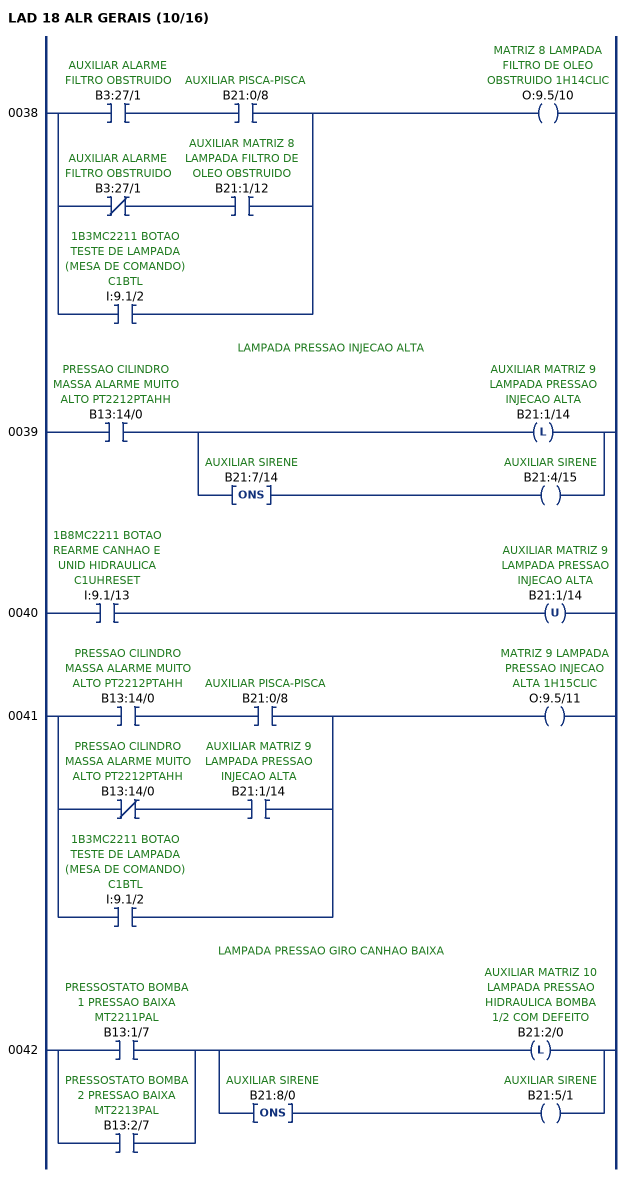
% Rung: 38 %
SOR BST XIC B3:27/1 XIC B21:0/8 NXB XIO B3:27/1 XIC B21:1/12 NXB XIC I:9.1/2 BND OTE O:9.5/10 EOR
%   B3:27/1  "AUXILIAR ALARME FILTRO OBSTRUIDO" %
%   B21:0/8  "AUXILIAR PISCA-PISCA" %
%   B21:1/12  "AUXILIAR MATRIZ 8 LAMPADA FILTRO DE OLEO OBSTRUIDO" %
%   I:9.1/2  C1BTL  "1B3MC2211 BOTAO TESTE DE LAMPADA (MESA DE COMANDO)" %
%   O:9.5/10  1H14CLIC  "MATRIZ 8 LAMPADA FILTRO DE OLEO OBSTRUIDO" %
% Rung: 39 %
% LAMPADA PRESSAO INJECAO ALTA %
SOR XIC B13:14/0 BST OTL B21:1/14 NXB OSR B21:7/14 OTE B21:4/15 BND EOR
%   B13:14/0  PT2212PTAHH  "PRESSAO CILINDRO MASSA ALARME MUITO ALTO" %
%   B21:1/14  "AUXILIAR MATRIZ 9 LAMPADA PRESSAO INJECAO ALTA" %
%   B21:7/14  "AUXILIAR SIRENE" %
%   B21:4/15  "AUXILIAR SIRENE" %
% Rung: 40 %
SOR XIC I:9.1/13 OTU B21:1/14 EOR
%   I:9.1/13  C1UHRESET  "1B8MC2211 BOTAO REARME CANHAO E UNID HIDRAULICA" %
%   B21:1/14  "AUXILIAR MATRIZ 9 LAMPADA PRESSAO INJECAO ALTA" %
% Rung: 41 %
SOR BST XIC B13:14/0 XIC B21:0/8 NXB XIO B13:14/0 XIC B21:1/14 NXB XIC I:9.1/2 BND OTE O:9.5/11 EOR
%   B13:14/0  PT2212PTAHH  "PRESSAO CILINDRO MASSA ALARME MUITO ALTO" %
%   B21:0/8  "AUXILIAR PISCA-PISCA" %
%   B21:1/14  "AUXILIAR MATRIZ 9 LAMPADA PRESSAO INJECAO ALTA" %
%   I:9.1/2  C1BTL  "1B3MC2211 BOTAO TESTE DE LAMPADA (MESA DE COMANDO)" %
%   O:9.5/11  1H15CLIC  "MATRIZ 9 LAMPADA PRESSAO INJECAO ALTA" %
% Rung: 42 %
% LAMPADA PRESSAO GIRO CANHAO BAIXA %
SOR BST XIC B13:1/7 NXB XIC B13:2/7 BND BST OTL B21:2/0 NXB OSR B21:8/0 OTE B21:5/1 BND EOR
%   B13:1/7  MT2211PAL  "PRESSOSTATO BOMBA 1 PRESSAO BAIXA" %
%   B13:2/7  MT2213PAL  "PRESSOSTATO BOMBA 2 PRESSAO BAIXA" %
%   B21:2/0  "AUXILIAR MATRIZ 10 LAMPADA PRESSAO HIDRAULICA BOMBA 1/2 COM DEFEITO" %
%   B21:8/0  "AUXILIAR SIRENE" %
%   B21:5/1  "AUXILIAR SIRENE" %

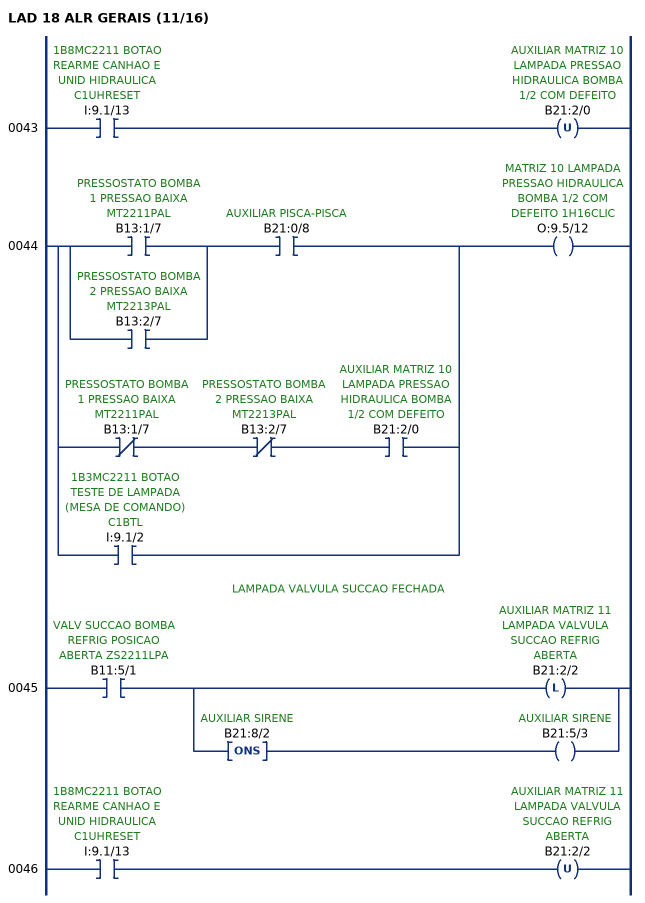
% Rung: 43 %
SOR XIC I:9.1/13 OTU B21:2/0 EOR
%   I:9.1/13  C1UHRESET  "1B8MC2211 BOTAO REARME CANHAO E UNID HIDRAULICA" %
%   B21:2/0  "AUXILIAR MATRIZ 10 LAMPADA PRESSAO HIDRAULICA BOMBA 1/2 COM DEFEITO" %
% Rung: 44 %
SOR BST BST XIC B13:1/7 NXB XIC B13:2/7 BND XIC B21:0/8 NXB XIO B13:1/7 XIO B13:2/7 XIC B21:2/0 NXB XIC I:9.1/2 BND OTE O:9.5/12 EOR
%   B13:1/7  MT2211PAL  "PRESSOSTATO BOMBA 1 PRESSAO BAIXA" %
%   B13:2/7  MT2213PAL  "PRESSOSTATO BOMBA 2 PRESSAO BAIXA" %
%   B21:0/8  "AUXILIAR PISCA-PISCA" %
%   B21:2/0  "AUXILIAR MATRIZ 10 LAMPADA PRESSAO HIDRAULICA BOMBA 1/2 COM DEFEITO" %
%   I:9.1/2  C1BTL  "1B3MC2211 BOTAO TESTE DE LAMPADA (MESA DE COMANDO)" %
%   O:9.5/12  1H16CLIC  "MATRIZ 10 LAMPADA PRESSAO HIDRAULICA BOMBA 1/2 COM DEFEITO" %
% Rung: 45 %
% LAMPADA VALVULA SUCCAO FECHADA %
SOR XIC B11:5/1 BST OTL B21:2/2 NXB OSR B21:8/2 OTE B21:5/3 BND EOR
%   B11:5/1  ZS2211LPA  "VALV SUCCAO BOMBA REFRIG POSICAO ABERTA" %
%   B21:2/2  "AUXILIAR MATRIZ 11 LAMPADA VALVULA SUCCAO REFRIG ABERTA" %
%   B21:8/2  "AUXILIAR SIRENE" %
%   B21:5/3  "AUXILIAR SIRENE" %
% Rung: 46 %
SOR XIC I:9.1/13 OTU B21:2/2 EOR
%   I:9.1/13  C1UHRESET  "1B8MC2211 BOTAO REARME CANHAO E UNID HIDRAULICA" %
%   B21:2/2  "AUXILIAR MATRIZ 11 LAMPADA VALVULA SUCCAO REFRIG ABERTA" %

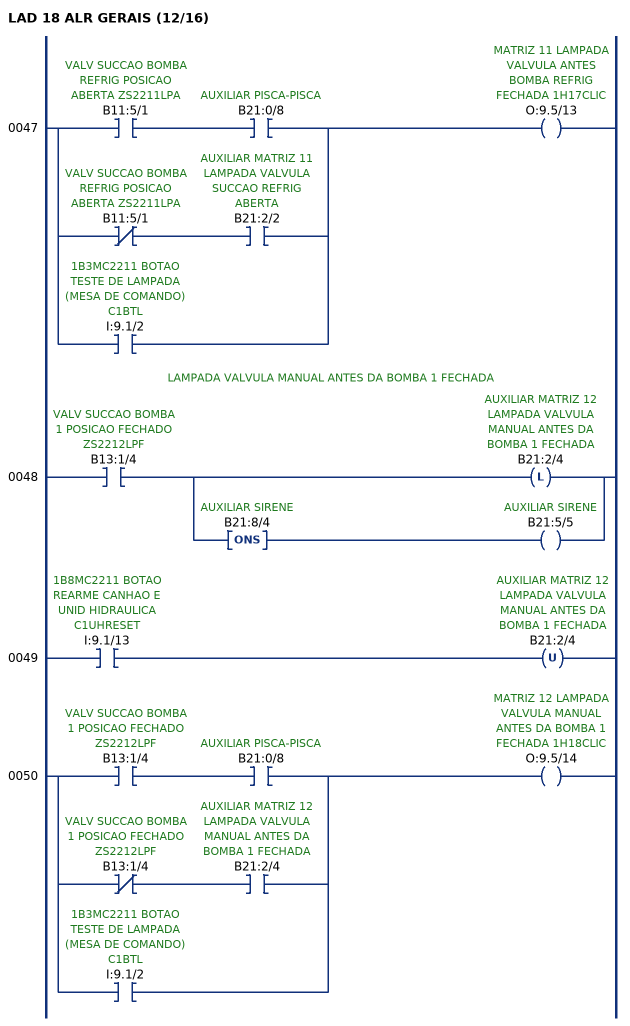
% Rung: 47 %
SOR BST XIC B11:5/1 XIC B21:0/8 NXB XIO B11:5/1 XIC B21:2/2 NXB XIC I:9.1/2 BND OTE O:9.5/13 EOR
%   B11:5/1  ZS2211LPA  "VALV SUCCAO BOMBA REFRIG POSICAO ABERTA" %
%   B21:0/8  "AUXILIAR PISCA-PISCA" %
%   B21:2/2  "AUXILIAR MATRIZ 11 LAMPADA VALVULA SUCCAO REFRIG ABERTA" %
%   I:9.1/2  C1BTL  "1B3MC2211 BOTAO TESTE DE LAMPADA (MESA DE COMANDO)" %
%   O:9.5/13  1H17CLIC  "MATRIZ 11 LAMPADA VALVULA ANTES BOMBA REFRIG FECHADA" %
% Rung: 48 %
% LAMPADA VALVULA MANUAL ANTES DA BOMBA 1 FECHADA %
SOR XIC B13:1/4 BST OTL B21:2/4 NXB OSR B21:8/4 OTE B21:5/5 BND EOR
%   B13:1/4  ZS2212LPF  "VALV SUCCAO BOMBA 1 POSICAO FECHADO" %
%   B21:2/4  "AUXILIAR MATRIZ 12 LAMPADA VALVULA MANUAL ANTES DA BOMBA 1 FECHADA" %
%   B21:8/4  "AUXILIAR SIRENE" %
%   B21:5/5  "AUXILIAR SIRENE" %
% Rung: 49 %
SOR XIC I:9.1/13 OTU B21:2/4 EOR
%   I:9.1/13  C1UHRESET  "1B8MC2211 BOTAO REARME CANHAO E UNID HIDRAULICA" %
%   B21:2/4  "AUXILIAR MATRIZ 12 LAMPADA VALVULA MANUAL ANTES DA BOMBA 1 FECHADA" %
% Rung: 50 %
SOR BST XIC B13:1/4 XIC B21:0/8 NXB XIO B13:1/4 XIC B21:2/4 NXB XIC I:9.1/2 BND OTE O:9.5/14 EOR
%   B13:1/4  ZS2212LPF  "VALV SUCCAO BOMBA 1 POSICAO FECHADO" %
%   B21:0/8  "AUXILIAR PISCA-PISCA" %
%   B21:2/4  "AUXILIAR MATRIZ 12 LAMPADA VALVULA MANUAL ANTES DA BOMBA 1 FECHADA" %
%   I:9.1/2  C1BTL  "1B3MC2211 BOTAO TESTE DE LAMPADA (MESA DE COMANDO)" %
%   O:9.5/14  1H18CLIC  "MATRIZ 12 LAMPADA VALVULA MANUAL ANTES DA BOMBA 1 FECHADA" %

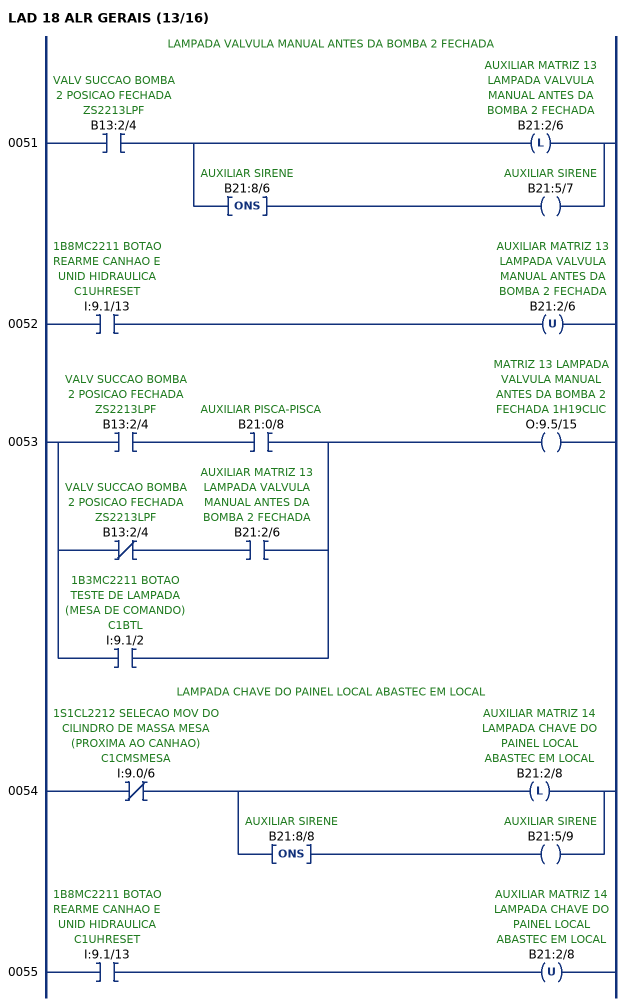
% Rung: 51 %
% LAMPADA VALVULA MANUAL ANTES DA BOMBA 2 FECHADA %
SOR XIC B13:2/4 BST OTL B21:2/6 NXB OSR B21:8/6 OTE B21:5/7 BND EOR
%   B13:2/4  ZS2213LPF  "VALV SUCCAO BOMBA 2 POSICAO FECHADA" %
%   B21:2/6  "AUXILIAR MATRIZ 13 LAMPADA VALVULA MANUAL ANTES DA BOMBA 2 FECHADA" %
%   B21:8/6  "AUXILIAR SIRENE" %
%   B21:5/7  "AUXILIAR SIRENE" %
% Rung: 52 %
SOR XIC I:9.1/13 OTU B21:2/6 EOR
%   I:9.1/13  C1UHRESET  "1B8MC2211 BOTAO REARME CANHAO E UNID HIDRAULICA" %
%   B21:2/6  "AUXILIAR MATRIZ 13 LAMPADA VALVULA MANUAL ANTES DA BOMBA 2 FECHADA" %
% Rung: 53 %
SOR BST XIC B13:2/4 XIC B21:0/8 NXB XIO B13:2/4 XIC B21:2/6 NXB XIC I:9.1/2 BND OTE O:9.5/15 EOR
%   B13:2/4  ZS2213LPF  "VALV SUCCAO BOMBA 2 POSICAO FECHADA" %
%   B21:0/8  "AUXILIAR PISCA-PISCA" %
%   B21:2/6  "AUXILIAR MATRIZ 13 LAMPADA VALVULA MANUAL ANTES DA BOMBA 2 FECHADA" %
%   I:9.1/2  C1BTL  "1B3MC2211 BOTAO TESTE DE LAMPADA (MESA DE COMANDO)" %
%   O:9.5/15  1H19CLIC  "MATRIZ 13 LAMPADA VALVULA MANUAL ANTES DA BOMBA 2 FECHADA" %
% Rung: 54 %
% LAMPADA CHAVE DO PAINEL LOCAL ABASTEC EM LOCAL %
SOR XIO I:9.0/6 BST OTL B21:2/8 NXB OSR B21:8/8 OTE B21:5/9 BND EOR
%   I:9.0/6  C1CMSMESA  "1S1CL2212 SELECAO MOV DO CILINDRO DE MASSA MESA (PROXIMA AO CANHAO)" %
%   B21:2/8  "AUXILIAR MATRIZ 14 LAMPADA CHAVE DO PAINEL LOCAL ABASTEC EM LOCAL" %
%   B21:8/8  "AUXILIAR SIRENE" %
%   B21:5/9  "AUXILIAR SIRENE" %
% Rung: 55 %
SOR XIC I:9.1/13 OTU B21:2/8 EOR
%   I:9.1/13  C1UHRESET  "1B8MC2211 BOTAO REARME CANHAO E UNID HIDRAULICA" %
%   B21:2/8  "AUXILIAR MATRIZ 14 LAMPADA CHAVE DO PAINEL LOCAL ABASTEC EM LOCAL" %

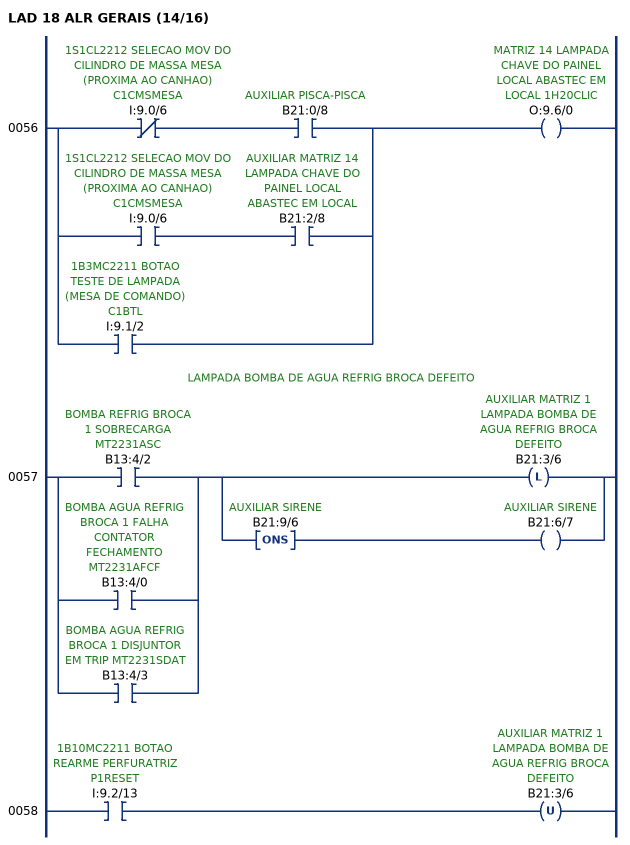
% Rung: 56 %
SOR BST XIO I:9.0/6 XIC B21:0/8 NXB XIC I:9.0/6 XIC B21:2/8 NXB XIC I:9.1/2 BND OTE O:9.6/0 EOR
%   I:9.0/6  C1CMSMESA  "1S1CL2212 SELECAO MOV DO CILINDRO DE MASSA MESA (PROXIMA AO CANHAO)" %
%   B21:0/8  "AUXILIAR PISCA-PISCA" %
%   B21:2/8  "AUXILIAR MATRIZ 14 LAMPADA CHAVE DO PAINEL LOCAL ABASTEC EM LOCAL" %
%   I:9.1/2  C1BTL  "1B3MC2211 BOTAO TESTE DE LAMPADA (MESA DE COMANDO)" %
%   O:9.6/0  1H20CLIC  "MATRIZ 14 LAMPADA CHAVE DO PAINEL LOCAL ABASTEC EM LOCAL" %
% Rung: 57 %
% LAMPADA BOMBA DE AGUA REFRIG BROCA DEFEITO %
SOR BST XIC B13:4/2 NXB XIC B13:4/0 NXB XIC B13:4/3 BND BST OTL B21:3/6 NXB OSR B21:9/6 OTE B21:6/7 BND EOR
%   B13:4/2  MT2231ASC  "BOMBA REFRIG BROCA 1 SOBRECARGA" %
%   B13:4/0  MT2231AFCF  "BOMBA AGUA REFRIG BROCA 1 FALHA CONTATOR FECHAMENTO" %
%   B13:4/3  MT2231SDAT  "BOMBA AGUA REFRIG BROCA 1 DISJUNTOR EM TRIP" %
%   B21:3/6  "AUXILIAR MATRIZ 1 LAMPADA BOMBA DE AGUA REFRIG BROCA DEFEITO" %
%   B21:9/6  "AUXILIAR SIRENE" %
%   B21:6/7  "AUXILIAR SIRENE" %
% Rung: 58 %
SOR XIC I:9.2/13 OTU B21:3/6 EOR
%   I:9.2/13  P1RESET  "1B10MC2211 BOTAO REARME PERFURATRIZ" %
%   B21:3/6  "AUXILIAR MATRIZ 1 LAMPADA BOMBA DE AGUA REFRIG BROCA DEFEITO" %

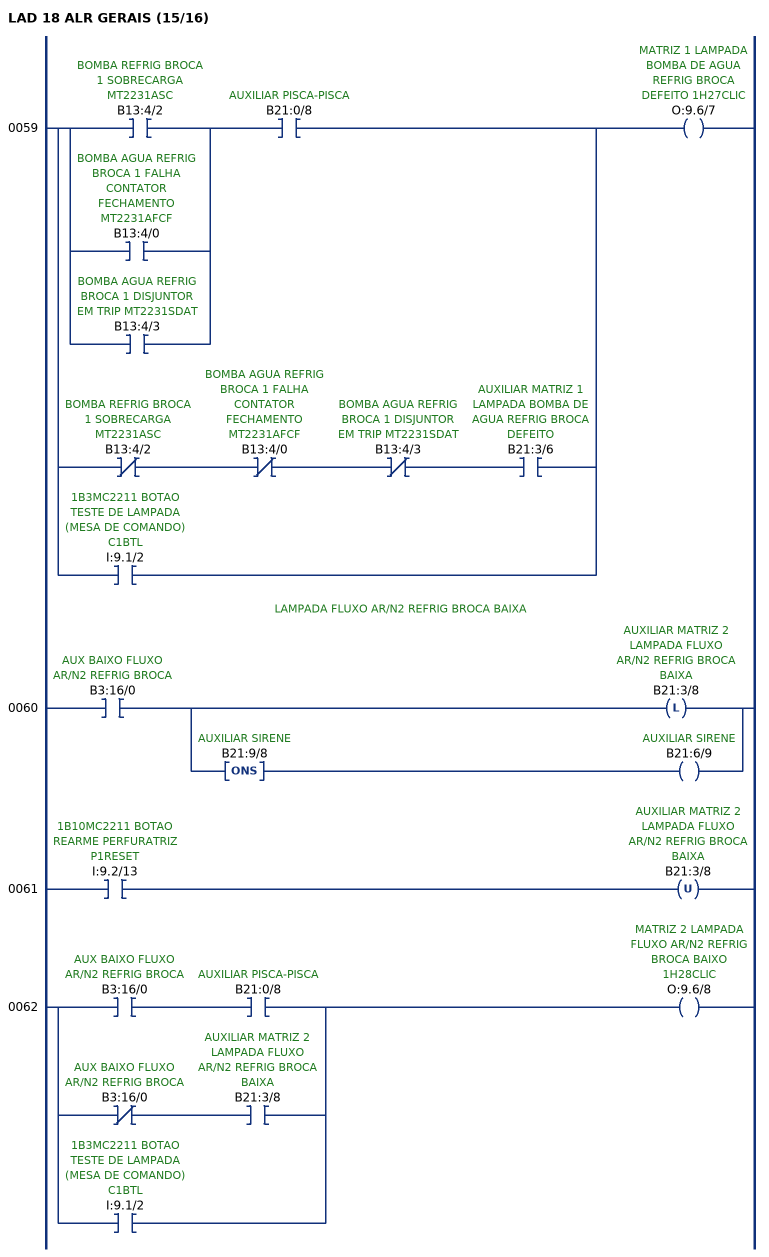
% Rung: 59 %
SOR BST BST XIC B13:4/2 NXB XIC B13:4/0 NXB XIC B13:4/3 BND XIC B21:0/8 NXB XIO B13:4/2 XIO B13:4/0 XIO B13:4/3 XIC B21:3/6 NXB XIC I:9.1/2 BND OTE O:9.6/7 EOR
%   B13:4/2  MT2231ASC  "BOMBA REFRIG BROCA 1 SOBRECARGA" %
%   B13:4/0  MT2231AFCF  "BOMBA AGUA REFRIG BROCA 1 FALHA CONTATOR FECHAMENTO" %
%   B13:4/3  MT2231SDAT  "BOMBA AGUA REFRIG BROCA 1 DISJUNTOR EM TRIP" %
%   B21:0/8  "AUXILIAR PISCA-PISCA" %
%   B21:3/6  "AUXILIAR MATRIZ 1 LAMPADA BOMBA DE AGUA REFRIG BROCA DEFEITO" %
%   I:9.1/2  C1BTL  "1B3MC2211 BOTAO TESTE DE LAMPADA (MESA DE COMANDO)" %
%   O:9.6/7  1H27CLIC  "MATRIZ 1 LAMPADA BOMBA DE AGUA REFRIG BROCA DEFEITO" %
% Rung: 60 %
% LAMPADA FLUXO AR/N2 REFRIG BROCA BAIXA %
SOR XIC B3:16/0 BST OTL B21:3/8 NXB OSR B21:9/8 OTE B21:6/9 BND EOR
%   B3:16/0  "AUX BAIXO FLUXO AR/N2 REFRIG BROCA" %
%   B21:3/8  "AUXILIAR MATRIZ 2 LAMPADA FLUXO AR/N2 REFRIG BROCA BAIXA" %
%   B21:9/8  "AUXILIAR SIRENE" %
%   B21:6/9  "AUXILIAR SIRENE" %
% Rung: 61 %
SOR XIC I:9.2/13 OTU B21:3/8 EOR
%   I:9.2/13  P1RESET  "1B10MC2211 BOTAO REARME PERFURATRIZ" %
%   B21:3/8  "AUXILIAR MATRIZ 2 LAMPADA FLUXO AR/N2 REFRIG BROCA BAIXA" %
% Rung: 62 %
SOR BST XIC B3:16/0 XIC B21:0/8 NXB XIO B3:16/0 XIC B21:3/8 NXB XIC I:9.1/2 BND OTE O:9.6/8 EOR
%   B3:16/0  "AUX BAIXO FLUXO AR/N2 REFRIG BROCA" %
%   B21:0/8  "AUXILIAR PISCA-PISCA" %
%   B21:3/8  "AUXILIAR MATRIZ 2 LAMPADA FLUXO AR/N2 REFRIG BROCA BAIXA" %
%   I:9.1/2  C1BTL  "1B3MC2211 BOTAO TESTE DE LAMPADA (MESA DE COMANDO)" %
%   O:9.6/8  1H28CLIC  "MATRIZ 2 LAMPADA FLUXO AR/N2 REFRIG BROCA BAIXO" %

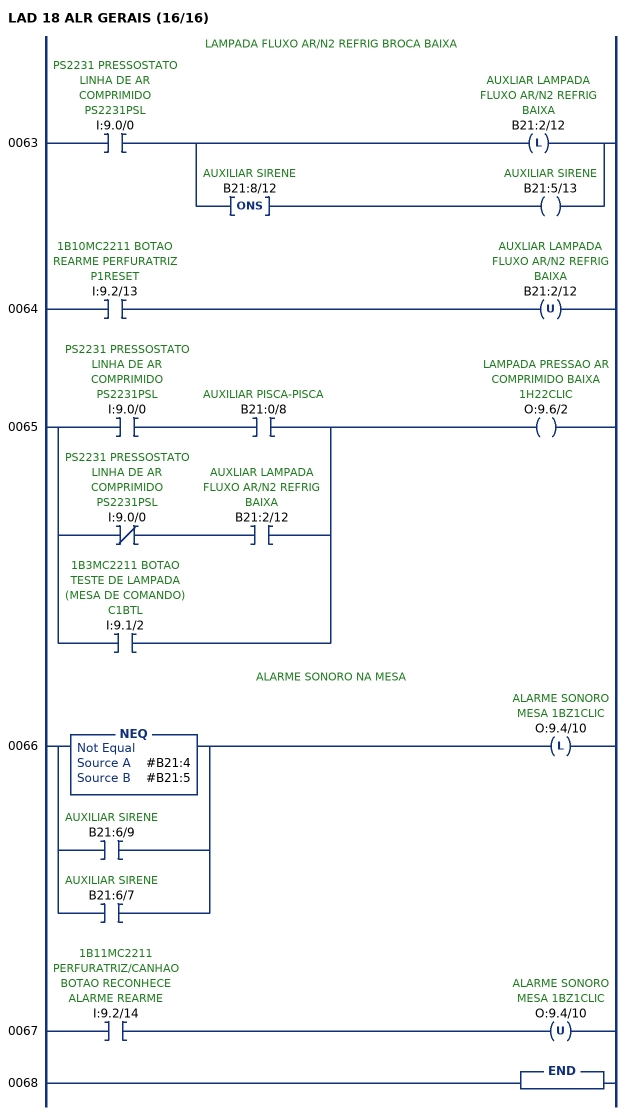
% Rung: 63 %
% LAMPADA FLUXO AR/N2 REFRIG BROCA BAIXA %
SOR XIC I:9.0/0 BST OTL B21:2/12 NXB OSR B21:8/12 OTE B21:5/13 BND EOR
%   I:9.0/0  PS2231PSL  "PS2231 PRESSOSTATO LINHA DE AR COMPRIMIDO" %
%   B21:2/12  "AUXLIAR LAMPADA FLUXO AR/N2 REFRIG BAIXA" %
%   B21:8/12  "AUXILIAR SIRENE" %
%   B21:5/13  "AUXILIAR SIRENE" %
% Rung: 64 %
SOR XIC I:9.2/13 OTU B21:2/12 EOR
%   I:9.2/13  P1RESET  "1B10MC2211 BOTAO REARME PERFURATRIZ" %
%   B21:2/12  "AUXLIAR LAMPADA FLUXO AR/N2 REFRIG BAIXA" %
% Rung: 65 %
SOR BST XIC I:9.0/0 XIC B21:0/8 NXB XIO I:9.0/0 XIC B21:2/12 NXB XIC I:9.1/2 BND OTE O:9.6/2 EOR
%   I:9.0/0  PS2231PSL  "PS2231 PRESSOSTATO LINHA DE AR COMPRIMIDO" %
%   B21:0/8  "AUXILIAR PISCA-PISCA" %
%   B21:2/12  "AUXLIAR LAMPADA FLUXO AR/N2 REFRIG BAIXA" %
%   I:9.1/2  C1BTL  "1B3MC2211 BOTAO TESTE DE LAMPADA (MESA DE COMANDO)" %
%   O:9.6/2  1H22CLIC  "LAMPADA PRESSAO AR COMPRIMIDO BAIXA" %
% Rung: 66 %
% ALARME SONORO NA MESA %
SOR BST NEQ #B21:4 #B21:5 NXB XIC B21:6/9 NXB XIC B21:6/7 BND OTL O:9.4/10 EOR
%   B21:6/9  "AUXILIAR SIRENE" %
%   B21:6/7  "AUXILIAR SIRENE" %
%   O:9.4/10  1BZ1CLIC  "ALARME SONORO MESA" %
% Rung: 67 %
SOR XIC I:9.2/14 OTU O:9.4/10 EOR
%   I:9.2/14  REARME  "1B11MC2211 PERFURATRIZ/CANHAO BOTAO RECONHECE ALARME" %
%   O:9.4/10  1BZ1CLIC  "ALARME SONORO MESA" %
% Rung: 68 %
SOR END EOR

LADDER 19 "COMUNIC"    % Comuinicao com supervisorio - Desabilitado(futuro) %
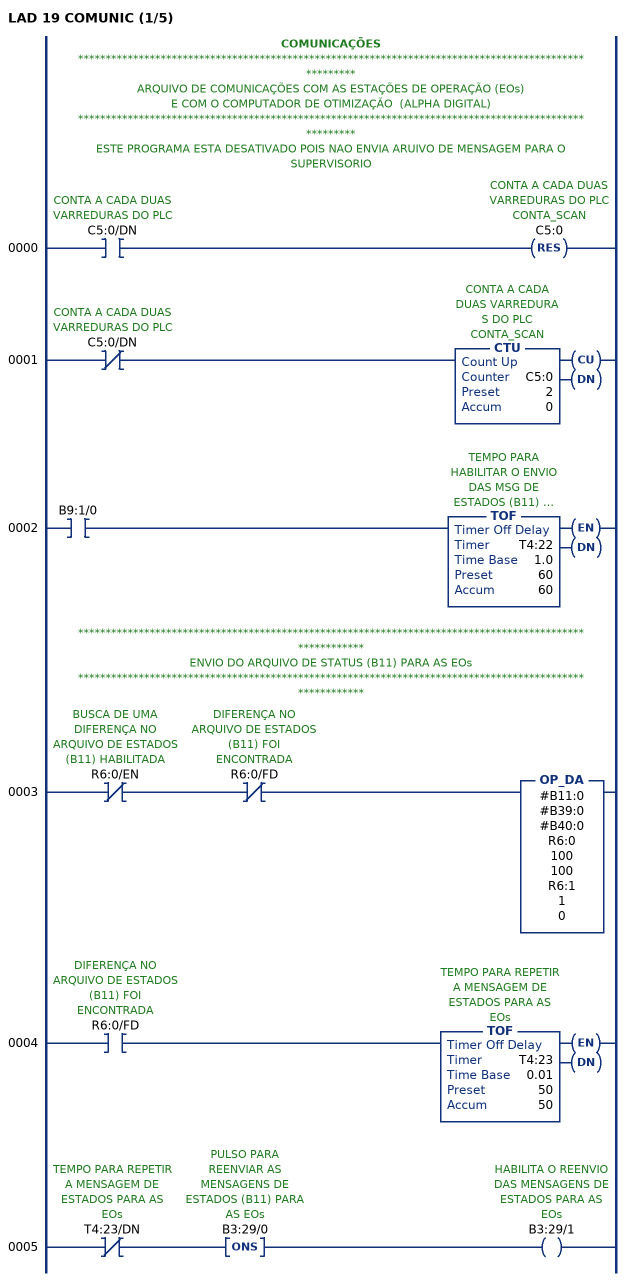
% Rung: 0 %
% TITLE: COMUNICAÇÕES %
% *****************************************************************************************************
% ARQUIVO DE COMUNICAÇÕES COM AS ESTAÇÕES DE OPERAÇÃO (EOs)
% E COM O COMPUTADOR DE OTIMIZAÇÃO  (ALPHA DIGITAL)
% *****************************************************************************************************
% ESTE PROGRAMA ESTA DESATIVADO POIS NAO ENVIA ARUIVO DE MENSAGEM PARA O SUPERVISORIO %
SOR XIC C5:0/DN RES C5:0 EOR
%   C5:0/DN  "CONTA A CADA DUAS VARREDURAS DO PLC" %
%   C5:0  CONTA_SCAN  "CONTA A CADA DUAS VARREDURAS DO PLC" %
% Rung: 1 %
SOR XIO C5:0/DN CTU C5:0 2 0 EOR
%   C5:0/DN  "CONTA A CADA DUAS VARREDURAS DO PLC" %
%   C5:0  CONTA_SCAN  "CONTA A CADA DUAS VARREDURAS DO PLC" %
% Rung: 2 %
SOR XIC B9:1/0 TOF T4:22 1.0 60 60 EOR
%   T4:22  "TEMPO PARA HABILITAR O ENVIO DAS MSG DE ESTADOS (B11) E DEFEITOS (B13) PARA A EO1" %
% Rung: 3 %
% ********************************************************************************************************
% ENVIO DO ARQUIVO DE STATUS (B11) PARA AS EOs
% ******************************************************************************************************** %
SOR XIO R6:0/EN XIO R6:0/FD OP_DA #B11:0 #B39:0 #B40:0 R6:0 100 100 R6:1 1 0 EOR
%   R6:0/EN  "BUSCA DE UMA DIFERENÇA NO ARQUIVO DE ESTADOS (B11) HABILITADA" %
%   R6:0/FD  "DIFERENÇA NO ARQUIVO DE ESTADOS (B11) FOI ENCONTRADA" %
%   B39:0  COPIA_DE_B11  "CÓPIA DO ARQUIVO DE ESTADOS (B11)" %
%   B40:0  RESULTADO_B11  "RESULTADO DA BUSCA DE DIFERENÇA NO ARQUIVO DE ESTADOS" %
%   R6:0  "BUSCA DE UMA DIFERENÇA NO ARQUIVO DE ESTADOS (B11)" %
% Rung: 4 %
SOR XIC R6:0/FD TOF T4:23 0.01 50 50 EOR
%   R6:0/FD  "DIFERENÇA NO ARQUIVO DE ESTADOS (B11) FOI ENCONTRADA" %
%   T4:23  "TEMPO PARA REPETIR A MENSAGEM DE ESTADOS PARA AS EOs" %
% Rung: 5 %
SOR XIO T4:23/DN OSR B3:29/0 OTE B3:29/1 EOR
%   T4:23  "TEMPO PARA REPETIR A MENSAGEM DE ESTADOS PARA AS EOs" %
%   B3:29/0  "PULSO PARA REENVIAR AS MENSAGENS DE ESTADOS (B11) PARA AS EOs" %
%   B3:29/1  "HABILITA O REENVIO DAS MENSAGENS DE ESTADOS PARA AS EOs" %

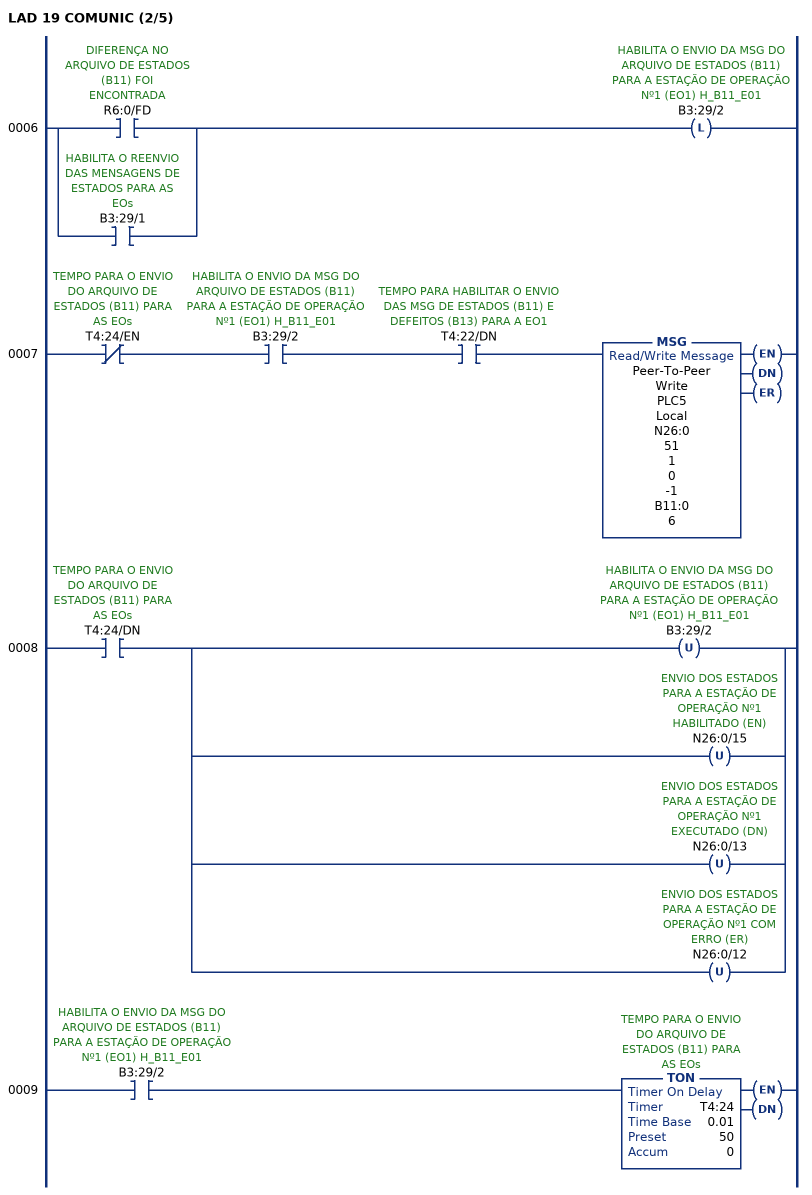
% Rung: 6 %
SOR BST XIC R6:0/FD NXB XIC B3:29/1 BND OTL B3:29/2 EOR
%   R6:0/FD  "DIFERENÇA NO ARQUIVO DE ESTADOS (B11) FOI ENCONTRADA" %
%   B3:29/1  "HABILITA O REENVIO DAS MENSAGENS DE ESTADOS PARA AS EOs" %
%   B3:29/2  H_B11_E01  "HABILITA O ENVIO DA MSG DO ARQUIVO DE ESTADOS (B11) PARA A ESTAÇÃO DE OPERAÇÃO Nº1 (EO1)" %
% Rung: 7 %
SOR XIO T4:24/EN XIC B3:29/2 XIC T4:22/DN MSG Peer-To-Peer Write PLC5 Local N26:0 51 1 0 -1 B11:0 6 EOR
%   T4:24  "TEMPO PARA O ENVIO DO ARQUIVO DE ESTADOS (B11) PARA AS EOs" %
%   B3:29/2  H_B11_E01  "HABILITA O ENVIO DA MSG DO ARQUIVO DE ESTADOS (B11) PARA A ESTAÇÃO DE OPERAÇÃO Nº1 (EO1)" %
%   T4:22  "TEMPO PARA HABILITAR O ENVIO DAS MSG DE ESTADOS (B11) E DEFEITOS (B13) PARA A EO1" %
%   MSG set-up: PLC5 Write | 5 | 6 | B11:0 | B11:0 | 0 | 0 | 0 | 100.100.100.1 | 0 | 0 %
%   N26:0  "ENVIO DOS ESTADOS PARA A ESTAÇÃO DE OPERAÇÃO Nº1" %
% Rung: 8 %
SOR XIC T4:24/DN BST OTU B3:29/2 NXB OTU N26:0/15 NXB OTU N26:0/13 NXB OTU N26:0/12 BND EOR
%   T4:24  "TEMPO PARA O ENVIO DO ARQUIVO DE ESTADOS (B11) PARA AS EOs" %
%   B3:29/2  H_B11_E01  "HABILITA O ENVIO DA MSG DO ARQUIVO DE ESTADOS (B11) PARA A ESTAÇÃO DE OPERAÇÃO Nº1 (EO1)" %
%   N26:0/15  "ENVIO DOS ESTADOS PARA A ESTAÇÃO DE OPERAÇÃO Nº1 HABILITADO (EN)" %
%   N26:0/13  "ENVIO DOS ESTADOS PARA A ESTAÇÃO DE OPERAÇÃO Nº1 EXECUTADO (DN)" %
%   N26:0/12  "ENVIO DOS ESTADOS PARA A ESTAÇÃO DE OPERAÇÃO Nº1 COM ERRO (ER)" %
% Rung: 9 %
SOR XIC B3:29/2 TON T4:24 0.01 50 0 EOR
%   B3:29/2  H_B11_E01  "HABILITA O ENVIO DA MSG DO ARQUIVO DE ESTADOS (B11) PARA A ESTAÇÃO DE OPERAÇÃO Nº1 (EO1)" %
%   T4:24  "TEMPO PARA O ENVIO DO ARQUIVO DE ESTADOS (B11) PARA AS EOs" %

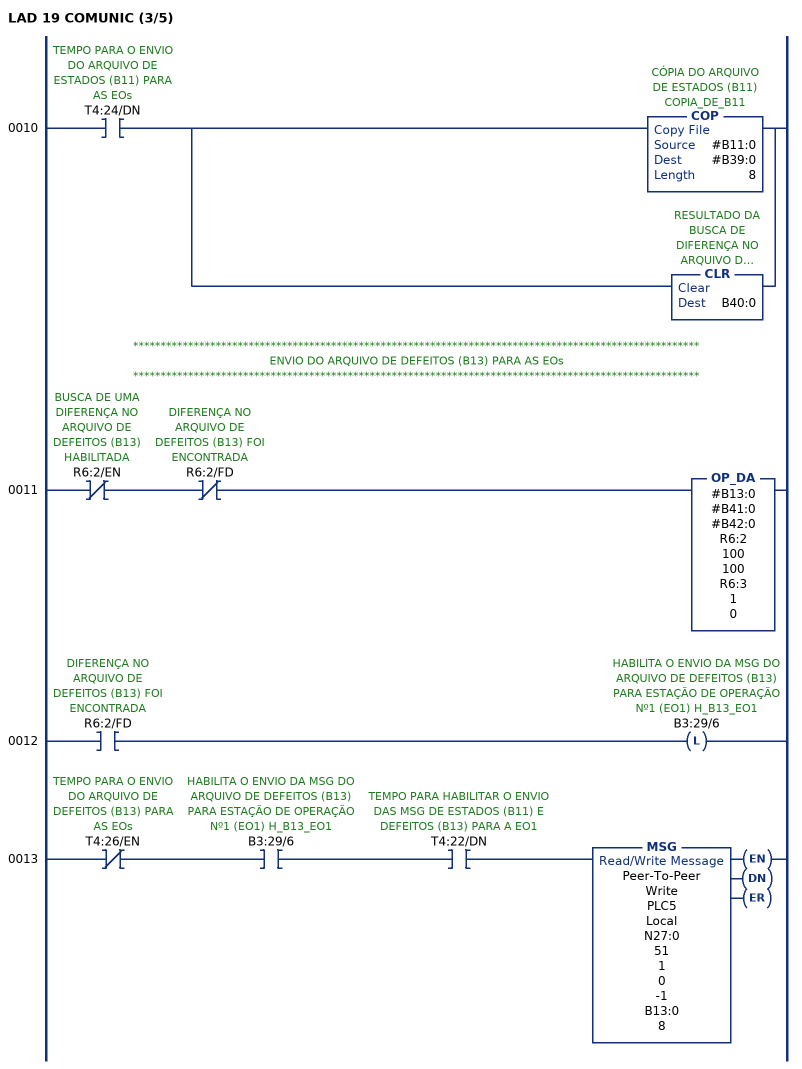
% Rung: 10 %
SOR XIC T4:24/DN BST COP #B11:0 #B39:0 8 NXB CLR B40:0 BND EOR
%   T4:24  "TEMPO PARA O ENVIO DO ARQUIVO DE ESTADOS (B11) PARA AS EOs" %
%   B39:0  COPIA_DE_B11  "CÓPIA DO ARQUIVO DE ESTADOS (B11)" %
%   B40:0  RESULTADO_B11  "RESULTADO DA BUSCA DE DIFERENÇA NO ARQUIVO DE ESTADOS" %
% Rung: 11 %
% *******************************************************************************************************
% ENVIO DO ARQUIVO DE DEFEITOS (B13) PARA AS EOs
% ******************************************************************************************************* %
SOR XIO R6:2/EN XIO R6:2/FD OP_DA #B13:0 #B41:0 #B42:0 R6:2 100 100 R6:3 1 0 EOR
%   R6:2/EN  "BUSCA DE UMA DIFERENÇA NO ARQUIVO DE DEFEITOS (B13) HABILITADA" %
%   R6:2/FD  "DIFERENÇA NO ARQUIVO DE DEFEITOS (B13) FOI ENCONTRADA" %
%   B41:0  COPIA_DE_B13  "CÓPIA DO ARQUIVO DE DEFEITOS (B13)" %
%   B42:0  RESULTADO_B13  "RESULTADO DA BUSCA DE DIFERENÇA NO ARQUIVO DE DEFEITOS (B13)" %
%   R6:2  "BUSCA DE UMA DIFERENÇA NO ARQUIVO DE DEFEITOS (B13)" %
% Rung: 12 %
SOR XIC R6:2/FD OTL B3:29/6 EOR
%   R6:2/FD  "DIFERENÇA NO ARQUIVO DE DEFEITOS (B13) FOI ENCONTRADA" %
%   B3:29/6  H_B13_EO1  "HABILITA O ENVIO DA MSG DO ARQUIVO DE DEFEITOS (B13) PARA ESTAÇÃO DE OPERAÇÃO Nº1 (EO1)" %
% Rung: 13 %
SOR XIO T4:26/EN XIC B3:29/6 XIC T4:22/DN MSG Peer-To-Peer Write PLC5 Local N27:0 51 1 0 -1 B13:0 8 EOR
%   T4:26  "TEMPO PARA O ENVIO DO ARQUIVO DE DEFEITOS (B13) PARA AS EOs" %
%   B3:29/6  H_B13_EO1  "HABILITA O ENVIO DA MSG DO ARQUIVO DE DEFEITOS (B13) PARA ESTAÇÃO DE OPERAÇÃO Nº1 (EO1)" %
%   T4:22  "TEMPO PARA HABILITAR O ENVIO DAS MSG DE ESTADOS (B11) E DEFEITOS (B13) PARA A EO1" %
%   MSG set-up: PLC5 Write | 5 | 8 | B13:0 | B13:0 | 0 | 0 | 0 | 100.100.100.1 | 0 | 0 %
%   N27:0  B13_EO1  "ENVIO DOS DEFEITOS PARA A ESTAÇÃO DE OPERAÇÃO Nº1" %

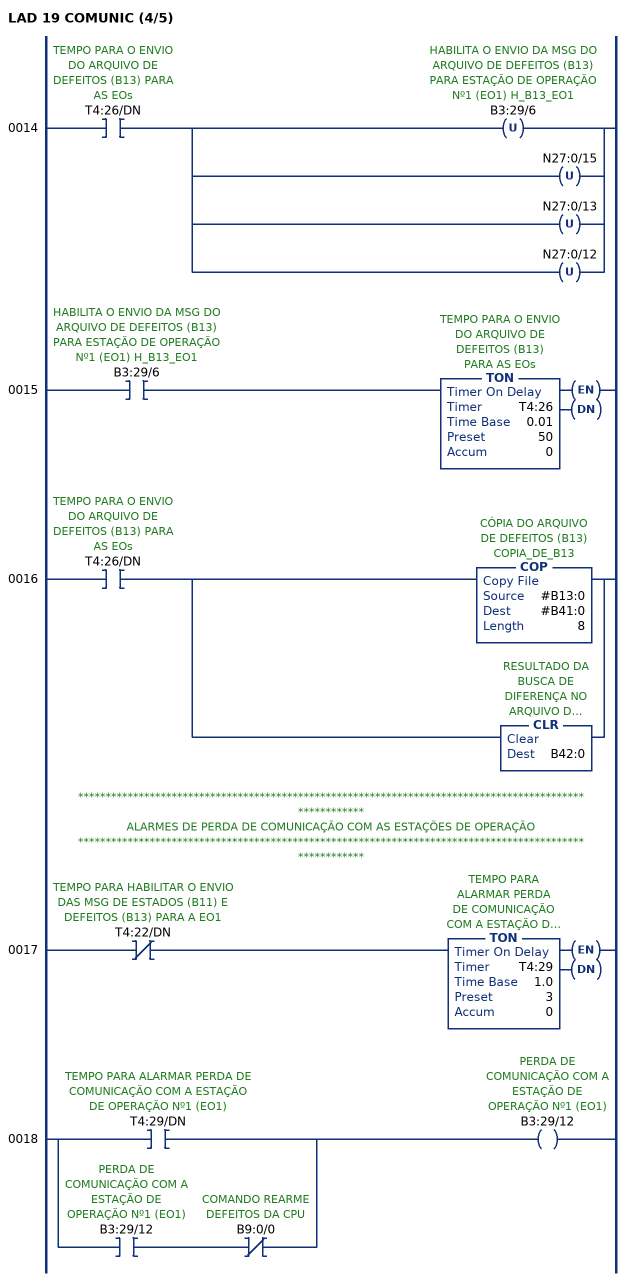
% Rung: 14 %
SOR XIC T4:26/DN BST OTU B3:29/6 NXB OTU N27:0/15 NXB OTU N27:0/13 NXB OTU N27:0/12 BND EOR
%   T4:26  "TEMPO PARA O ENVIO DO ARQUIVO DE DEFEITOS (B13) PARA AS EOs" %
%   B3:29/6  H_B13_EO1  "HABILITA O ENVIO DA MSG DO ARQUIVO DE DEFEITOS (B13) PARA ESTAÇÃO DE OPERAÇÃO Nº1 (EO1)" %
% Rung: 15 %
SOR XIC B3:29/6 TON T4:26 0.01 50 0 EOR
%   B3:29/6  H_B13_EO1  "HABILITA O ENVIO DA MSG DO ARQUIVO DE DEFEITOS (B13) PARA ESTAÇÃO DE OPERAÇÃO Nº1 (EO1)" %
%   T4:26  "TEMPO PARA O ENVIO DO ARQUIVO DE DEFEITOS (B13) PARA AS EOs" %
% Rung: 16 %
SOR XIC T4:26/DN BST COP #B13:0 #B41:0 8 NXB CLR B42:0 BND EOR
%   T4:26  "TEMPO PARA O ENVIO DO ARQUIVO DE DEFEITOS (B13) PARA AS EOs" %
%   B41:0  COPIA_DE_B13  "CÓPIA DO ARQUIVO DE DEFEITOS (B13)" %
%   B42:0  RESULTADO_B13  "RESULTADO DA BUSCA DE DIFERENÇA NO ARQUIVO DE DEFEITOS (B13)" %
% Rung: 17 %
% ********************************************************************************************************
% ALARMES DE PERDA DE COMUNICAÇÃO COM AS ESTAÇÕES DE OPERAÇÃO
% ******************************************************************************************************** %
SOR XIO T4:22/DN TON T4:29 1.0 3 0 EOR
%   T4:22  "TEMPO PARA HABILITAR O ENVIO DAS MSG DE ESTADOS (B11) E DEFEITOS (B13) PARA A EO1" %
%   T4:29  "TEMPO PARA ALARMAR PERDA DE COMUNICAÇÃO COM A ESTAÇÃO DE OPERAÇÃO Nº1 (EO1)" %
% Rung: 18 %
SOR BST XIC T4:29/DN NXB XIC B3:29/12 XIO B9:0/0 BND OTE B3:29/12 EOR
%   T4:29  "TEMPO PARA ALARMAR PERDA DE COMUNICAÇÃO COM A ESTAÇÃO DE OPERAÇÃO Nº1 (EO1)" %
%   B3:29/12  "PERDA DE COMUNICAÇÃO COM A ESTAÇÃO DE OPERAÇÃO Nº1 (EO1)" %
%   B9:0/0  "COMANDO REARME DEFEITOS DA CPU" %

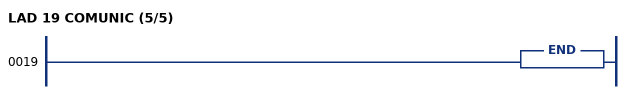
% Rung: 19 %
SOR END EOR

LADDER 20 "HISTERESE"
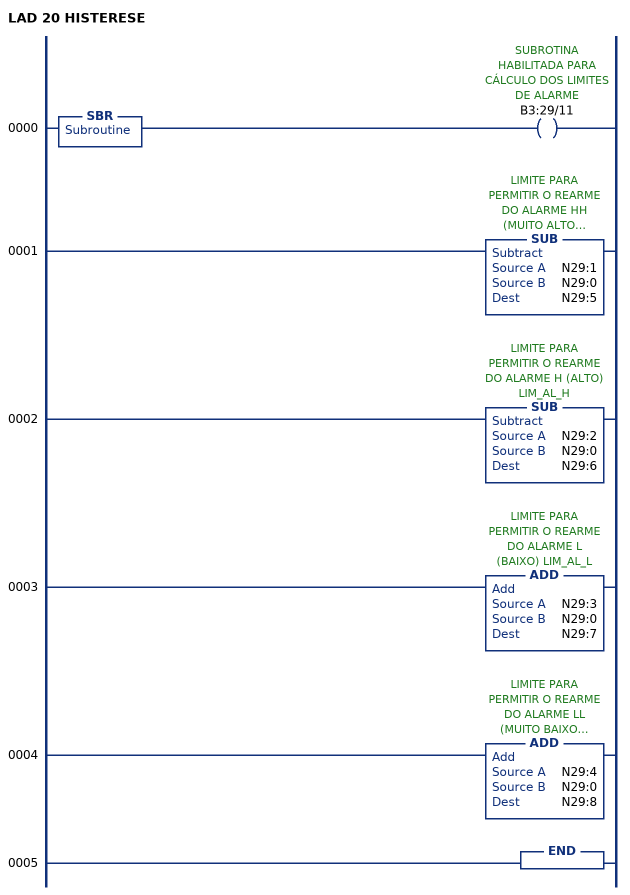
% Rung: 0 %
SOR SBR OTE B3:29/11 EOR
%   B3:29/11  "SUBROTINA HABILITADA PARA CÁLCULO DOS LIMITES DE ALARME" %
% Rung: 1 %
SOR SUB N29:1 N29:0 N29:5 EOR
%   N29:1  ALARME_HH %
%   N29:0  HISTERESE  "VALOR DE HISTERESE PARA CÁLCULO DOS ALARMES ANALÓGICOS" %
%   N29:5  LIM_AL_HH  "LIMITE PARA PERMITIR O REARME DO ALARME HH (MUITO ALTO)" %
% Rung: 2 %
SOR SUB N29:2 N29:0 N29:6 EOR
%   N29:2  ALARME_H %
%   N29:0  HISTERESE  "VALOR DE HISTERESE PARA CÁLCULO DOS ALARMES ANALÓGICOS" %
%   N29:6  LIM_AL_H  "LIMITE PARA PERMITIR O REARME DO ALARME H (ALTO)" %
% Rung: 3 %
SOR ADD N29:3 N29:0 N29:7 EOR
%   N29:3  ALARME_L %
%   N29:0  HISTERESE  "VALOR DE HISTERESE PARA CÁLCULO DOS ALARMES ANALÓGICOS" %
%   N29:7  LIM_AL_L  "LIMITE PARA PERMITIR O REARME DO ALARME L (BAIXO)" %
% Rung: 4 %
SOR ADD N29:4 N29:0 N29:8 EOR
%   N29:4  ALARME_LL %
%   N29:0  HISTERESE  "VALOR DE HISTERESE PARA CÁLCULO DOS ALARMES ANALÓGICOS" %
%   N29:8  LIM_AL_LL  "LIMITE PARA PERMITIR O REARME DO ALARME LL (MUITO BAIXO)" %
% Rung: 5 %
SOR END EOR

LADDER 21 "ALR ANALOG"    % Alarmes Analogicos %
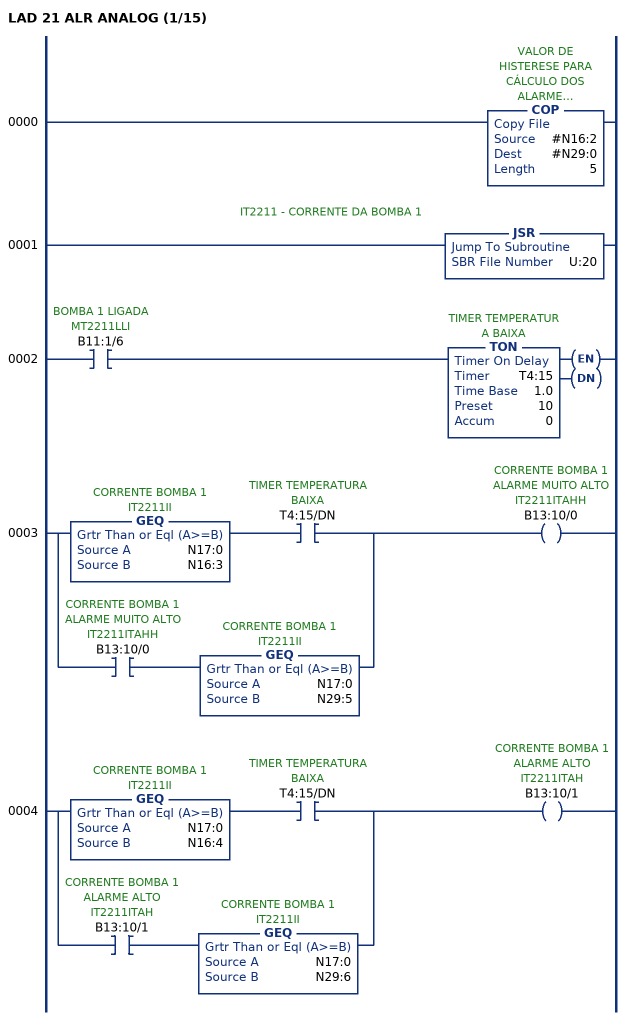
% Rung: 0 %
SOR COP #N16:2 #N29:0 5 EOR
%   N16:2  IT2211HIS  "CORRENTE BOMBA 1 HISTERESE" %
%   N29:0  HISTERESE  "VALOR DE HISTERESE PARA CÁLCULO DOS ALARMES ANALÓGICOS" %
% Rung: 1 %
% IT2211 - CORRENTE DA BOMBA 1 %
SOR JSR U:20 EOR
% Rung: 2 %
SOR XIC B11:1/6 TON T4:15 1.0 10 0 EOR
%   B11:1/6  MT2211LLI  "BOMBA 1 LIGADA" %
%   T4:15  "TIMER TEMPERATURA BAIXA" %
% Rung: 3 %
SOR BST GEQ N17:0 N16:3 XIC T4:15/DN NXB XIC B13:10/0 GEQ N17:0 N29:5 BND OTE B13:10/0 EOR
%   N17:0  IT2211II  "CORRENTE BOMBA 1" %
%   N16:3  IT2211HH  "CORRENTE BOMBA 1 MUITO ALTA" %
%   T4:15  "TIMER TEMPERATURA BAIXA" %
%   B13:10/0  IT2211ITAHH  "CORRENTE BOMBA 1 ALARME MUITO ALTO" %
%   N29:5  LIM_AL_HH  "LIMITE PARA PERMITIR O REARME DO ALARME HH (MUITO ALTO)" %
% Rung: 4 %
SOR BST GEQ N17:0 N16:4 XIC T4:15/DN NXB XIC B13:10/1 GEQ N17:0 N29:6 BND OTE B13:10/1 EOR
%   N17:0  IT2211II  "CORRENTE BOMBA 1" %
%   N16:4  IT2211H  "CORRENTE BOMBA 1 ALTA" %
%   T4:15  "TIMER TEMPERATURA BAIXA" %
%   B13:10/1  IT2211ITAH  "CORRENTE BOMBA 1 ALARME ALTO" %
%   N29:6  LIM_AL_H  "LIMITE PARA PERMITIR O REARME DO ALARME H (ALTO)" %

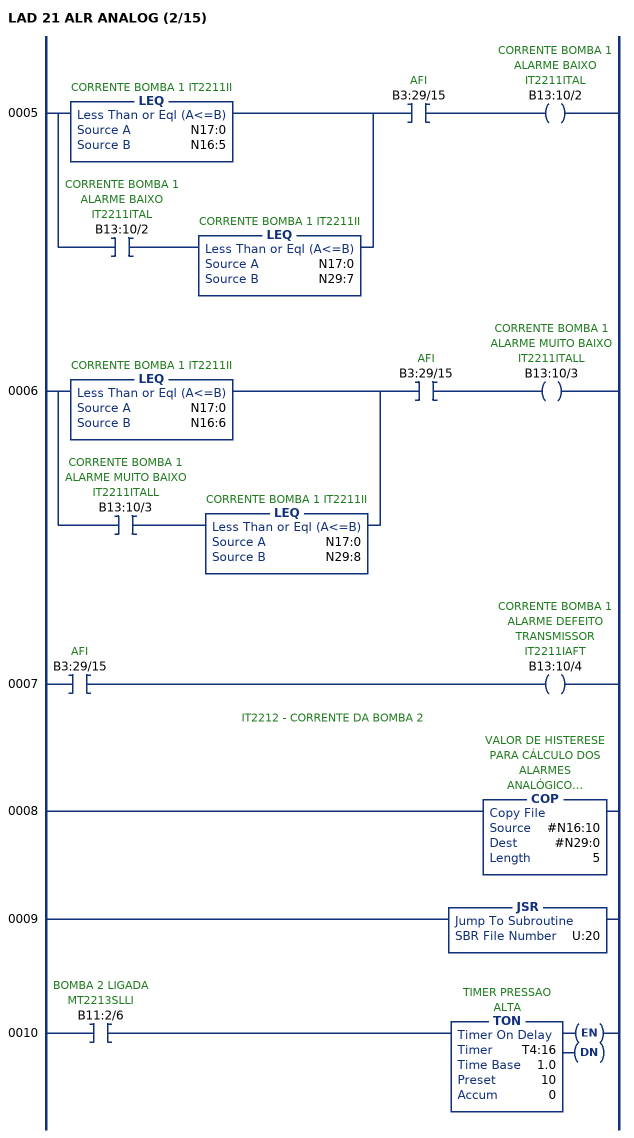
% Rung: 5 %
SOR BST LEQ N17:0 N16:5 NXB XIC B13:10/2 LEQ N17:0 N29:7 BND XIC B3:29/15 OTE B13:10/2 EOR
%   N17:0  IT2211II  "CORRENTE BOMBA 1" %
%   N16:5  IT2211L  "CORRENTE BOMBA 1 BAIXA" %
%   B13:10/2  IT2211ITAL  "CORRENTE BOMBA 1 ALARME BAIXO" %
%   N29:7  LIM_AL_L  "LIMITE PARA PERMITIR O REARME DO ALARME L (BAIXO)" %
%   B3:29/15  AFI %
% Rung: 6 %
SOR BST LEQ N17:0 N16:6 NXB XIC B13:10/3 LEQ N17:0 N29:8 BND XIC B3:29/15 OTE B13:10/3 EOR
%   N17:0  IT2211II  "CORRENTE BOMBA 1" %
%   N16:6  IT2211LL  "CORRENTE BOMBA 1 MUITO BAIXA" %
%   B13:10/3  IT2211ITALL  "CORRENTE BOMBA 1 ALARME MUITO BAIXO" %
%   N29:8  LIM_AL_LL  "LIMITE PARA PERMITIR O REARME DO ALARME LL (MUITO BAIXO)" %
%   B3:29/15  AFI %
% Rung: 7 %
SOR XIC B3:29/15 OTE B13:10/4 EOR
%   B3:29/15  AFI %
%   B13:10/4  IT2211IAFT  "CORRENTE BOMBA 1 ALARME DEFEITO TRANSMISSOR" %
% Rung: 8 %
% IT2212 - CORRENTE DA BOMBA 2 %
SOR COP #N16:10 #N29:0 5 EOR
%   N16:10  IT2212HIS  "CORRENTE BOMBA 2 HISTERESE" %
%   N29:0  HISTERESE  "VALOR DE HISTERESE PARA CÁLCULO DOS ALARMES ANALÓGICOS" %
% Rung: 9 %
SOR JSR U:20 EOR
% Rung: 10 %
SOR XIC B11:2/6 TON T4:16 1.0 10 0 EOR
%   B11:2/6  MT2213SLLI  "BOMBA 2 LIGADA" %
%   T4:16  "TIMER PRESSAO ALTA" %

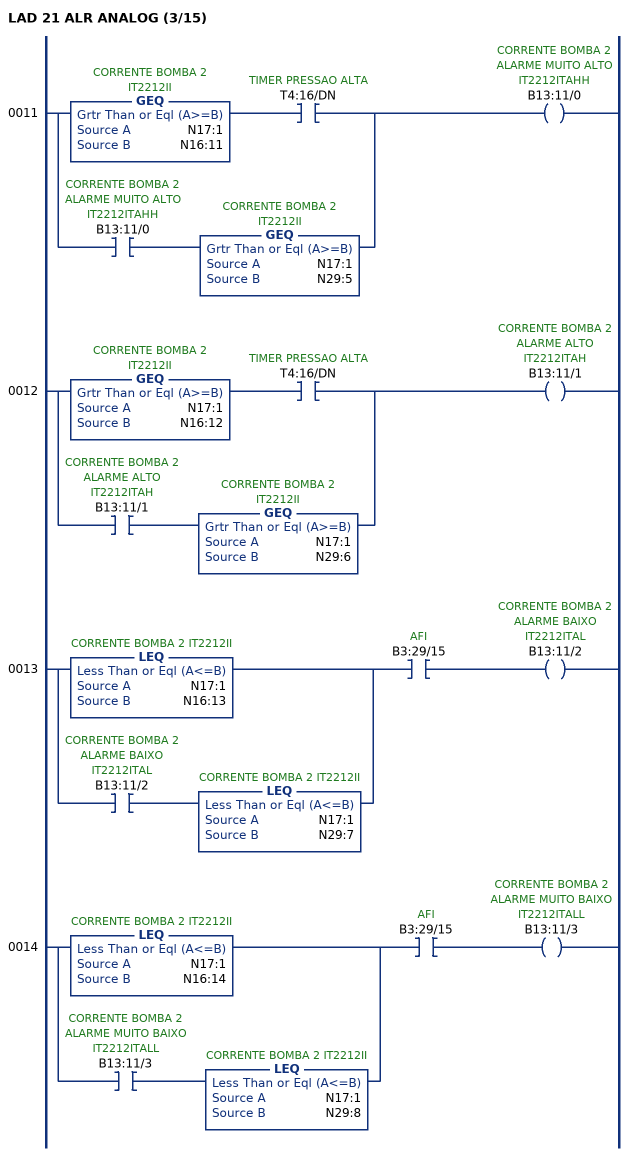
% Rung: 11 %
SOR BST GEQ N17:1 N16:11 XIC T4:16/DN NXB XIC B13:11/0 GEQ N17:1 N29:5 BND OTE B13:11/0 EOR
%   N17:1  IT2212II  "CORRENTE BOMBA 2" %
%   N16:11  IT2212HH  "CORRENTE BOMBA 2 MUITO ALTA" %
%   T4:16  "TIMER PRESSAO ALTA" %
%   B13:11/0  IT2212ITAHH  "CORRENTE BOMBA 2 ALARME MUITO ALTO" %
%   N29:5  LIM_AL_HH  "LIMITE PARA PERMITIR O REARME DO ALARME HH (MUITO ALTO)" %
% Rung: 12 %
SOR BST GEQ N17:1 N16:12 XIC T4:16/DN NXB XIC B13:11/1 GEQ N17:1 N29:6 BND OTE B13:11/1 EOR
%   N17:1  IT2212II  "CORRENTE BOMBA 2" %
%   N16:12  IT2212H  "CORRENTE BOMBA 2 ALTA" %
%   T4:16  "TIMER PRESSAO ALTA" %
%   B13:11/1  IT2212ITAH  "CORRENTE BOMBA 2 ALARME ALTO" %
%   N29:6  LIM_AL_H  "LIMITE PARA PERMITIR O REARME DO ALARME H (ALTO)" %
% Rung: 13 %
SOR BST LEQ N17:1 N16:13 NXB XIC B13:11/2 LEQ N17:1 N29:7 BND XIC B3:29/15 OTE B13:11/2 EOR
%   N17:1  IT2212II  "CORRENTE BOMBA 2" %
%   N16:13  IT2212L  "CORRENTE BOMBA 2 BAIXA" %
%   B13:11/2  IT2212ITAL  "CORRENTE BOMBA 2 ALARME BAIXO" %
%   N29:7  LIM_AL_L  "LIMITE PARA PERMITIR O REARME DO ALARME L (BAIXO)" %
%   B3:29/15  AFI %
% Rung: 14 %
SOR BST LEQ N17:1 N16:14 NXB XIC B13:11/3 LEQ N17:1 N29:8 BND XIC B3:29/15 OTE B13:11/3 EOR
%   N17:1  IT2212II  "CORRENTE BOMBA 2" %
%   N16:14  IT2212LL  "CORRENTE BOMBA 2 MUITO BAIXA" %
%   B13:11/3  IT2212ITALL  "CORRENTE BOMBA 2 ALARME MUITO BAIXO" %
%   N29:8  LIM_AL_LL  "LIMITE PARA PERMITIR O REARME DO ALARME LL (MUITO BAIXO)" %
%   B3:29/15  AFI %

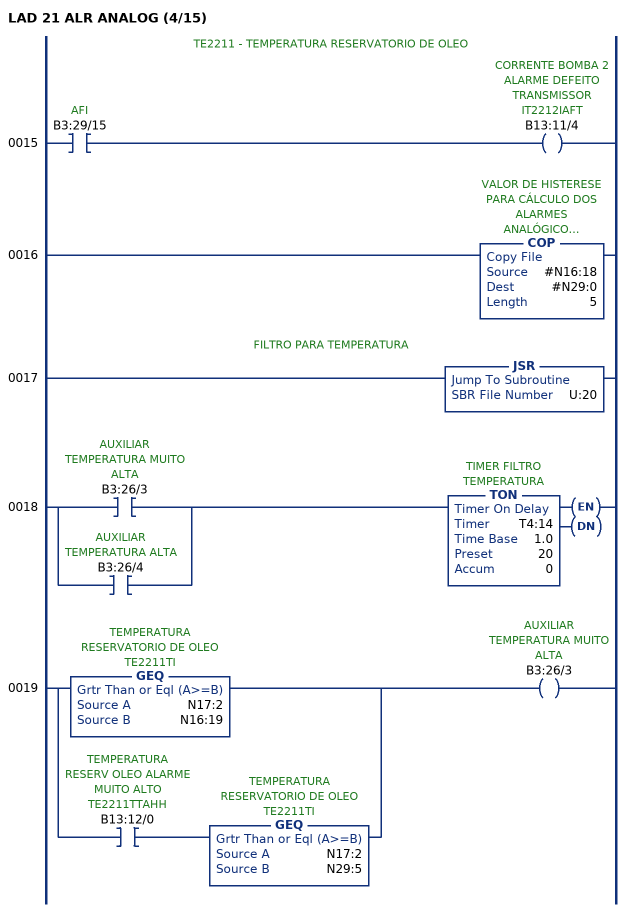
% Rung: 15 %
% TE2211 - TEMPERATURA RESERVATORIO DE OLEO %
SOR XIC B3:29/15 OTE B13:11/4 EOR
%   B3:29/15  AFI %
%   B13:11/4  IT2212IAFT  "CORRENTE BOMBA 2 ALARME DEFEITO TRANSMISSOR" %
% Rung: 16 %
SOR COP #N16:18 #N29:0 5 EOR
%   N16:18  TE2211HIS  "TEMPERATURA RESERVATORIO DE OLEO HISTERESE" %
%   N29:0  HISTERESE  "VALOR DE HISTERESE PARA CÁLCULO DOS ALARMES ANALÓGICOS" %
% Rung: 17 %
% FILTRO PARA TEMPERATURA %
SOR JSR U:20 EOR
% Rung: 18 %
SOR BST XIC B3:26/3 NXB XIC B3:26/4 BND TON T4:14 1.0 20 0 EOR
%   B3:26/3  "AUXILIAR TEMPERATURA MUITO ALTA" %
%   B3:26/4  "AUXILIAR TEMPERATURA ALTA" %
%   T4:14  "TIMER FILTRO TEMPERATURA" %
% Rung: 19 %
SOR BST GEQ N17:2 N16:19 NXB XIC B13:12/0 GEQ N17:2 N29:5 BND OTE B3:26/3 EOR
%   N17:2  TE2211TI  "TEMPERATURA RESERVATORIO DE OLEO" %
%   N16:19  TE2211HH  "TEMPERATURA RESERVATORIO DE OLEO MUITO ALTA" %
%   B13:12/0  TE2211TTAHH  "TEMPERATURA RESERV OLEO ALARME MUITO ALTO" %
%   N29:5  LIM_AL_HH  "LIMITE PARA PERMITIR O REARME DO ALARME HH (MUITO ALTO)" %
%   B3:26/3  "AUXILIAR TEMPERATURA MUITO ALTA" %

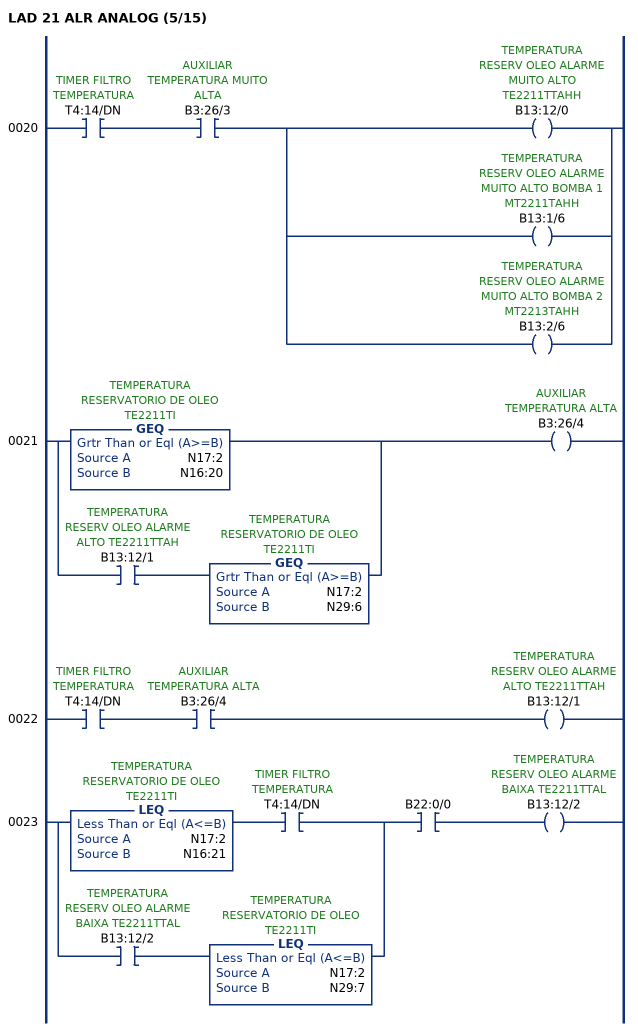
% Rung: 20 %
SOR XIC T4:14/DN XIC B3:26/3 BST OTE B13:12/0 NXB OTE B13:1/6 NXB OTE B13:2/6 BND EOR
%   T4:14  "TIMER FILTRO TEMPERATURA" %
%   B3:26/3  "AUXILIAR TEMPERATURA MUITO ALTA" %
%   B13:12/0  TE2211TTAHH  "TEMPERATURA RESERV OLEO ALARME MUITO ALTO" %
%   B13:1/6  MT2211TAHH  "TEMPERATURA RESERV OLEO ALARME MUITO ALTO BOMBA 1" %
%   B13:2/6  MT2213TAHH  "TEMPERATURA RESERV OLEO ALARME MUITO ALTO BOMBA 2" %
% Rung: 21 %
SOR BST GEQ N17:2 N16:20 NXB XIC B13:12/1 GEQ N17:2 N29:6 BND OTE B3:26/4 EOR
%   N17:2  TE2211TI  "TEMPERATURA RESERVATORIO DE OLEO" %
%   N16:20  TE2211H  "TEMPERATURA RESERVATORIO DE OLEO ALTA" %
%   B13:12/1  TE2211TTAH  "TEMPERATURA RESERV OLEO ALARME ALTO" %
%   N29:6  LIM_AL_H  "LIMITE PARA PERMITIR O REARME DO ALARME H (ALTO)" %
%   B3:26/4  "AUXILIAR TEMPERATURA ALTA" %
% Rung: 22 %
SOR XIC T4:14/DN XIC B3:26/4 OTE B13:12/1 EOR
%   T4:14  "TIMER FILTRO TEMPERATURA" %
%   B3:26/4  "AUXILIAR TEMPERATURA ALTA" %
%   B13:12/1  TE2211TTAH  "TEMPERATURA RESERV OLEO ALARME ALTO" %
% Rung: 23 %
SOR BST LEQ N17:2 N16:21 XIC T4:14/DN NXB XIC B13:12/2 LEQ N17:2 N29:7 BND XIC B22:0/0 OTE B13:12/2 EOR
%   N17:2  TE2211TI  "TEMPERATURA RESERVATORIO DE OLEO" %
%   N16:21  TE2211L  "TEMPERATURA RESERVATORIO DE OLEO BAIXA" %
%   T4:14  "TIMER FILTRO TEMPERATURA" %
%   B13:12/2  TE2211TTAL  "TEMPERATURA RESERV OLEO ALARME BAIXA" %
%   N29:7  LIM_AL_L  "LIMITE PARA PERMITIR O REARME DO ALARME L (BAIXO)" %

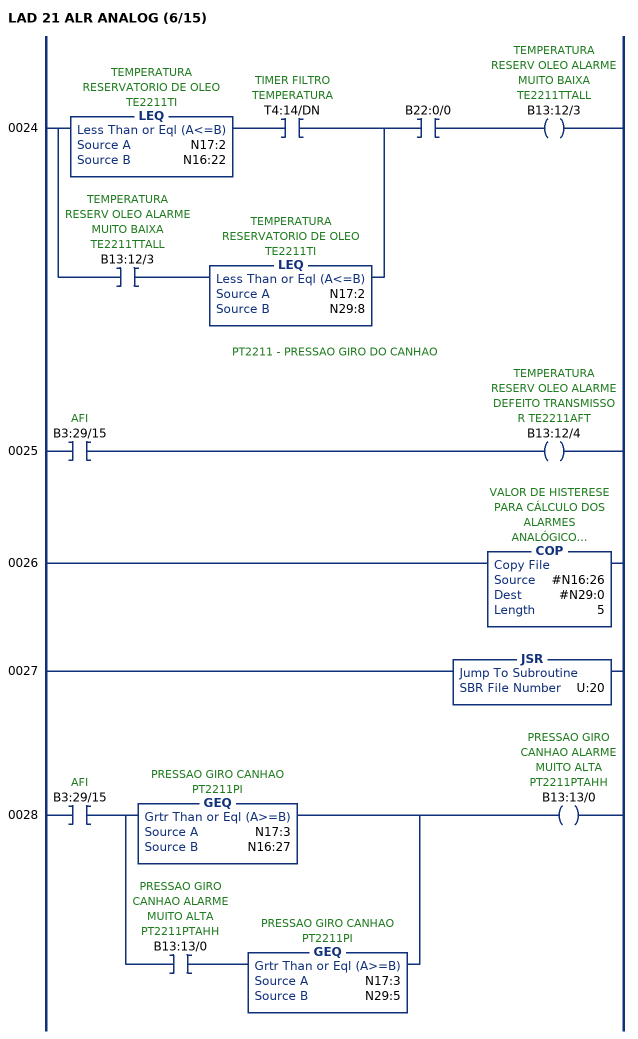
% Rung: 24 %
SOR BST LEQ N17:2 N16:22 XIC T4:14/DN NXB XIC B13:12/3 LEQ N17:2 N29:8 BND XIC B22:0/0 OTE B13:12/3 EOR
%   N17:2  TE2211TI  "TEMPERATURA RESERVATORIO DE OLEO" %
%   N16:22  TE2211LL  "TEMPERATURA RESERVATORIO DE OLEO MUITO BAIXA" %
%   T4:14  "TIMER FILTRO TEMPERATURA" %
%   B13:12/3  TE2211TTALL  "TEMPERATURA RESERV OLEO ALARME MUITO BAIXA" %
%   N29:8  LIM_AL_LL  "LIMITE PARA PERMITIR O REARME DO ALARME LL (MUITO BAIXO)" %
% Rung: 25 %
% PT2211 - PRESSAO GIRO DO CANHAO %
SOR XIC B3:29/15 OTE B13:12/4 EOR
%   B3:29/15  AFI %
%   B13:12/4  TE2211AFT  "TEMPERATURA RESERV OLEO ALARME DEFEITO TRANSMISSOR" %
% Rung: 26 %
SOR COP #N16:26 #N29:0 5 EOR
%   N16:26  PT2211HIS  "GIRO CANHAO PRESSAO HISTERESE" %
%   N29:0  HISTERESE  "VALOR DE HISTERESE PARA CÁLCULO DOS ALARMES ANALÓGICOS" %
% Rung: 27 %
SOR JSR U:20 EOR
% Rung: 28 %
SOR XIC B3:29/15 BST GEQ N17:3 N16:27 NXB XIC B13:13/0 GEQ N17:3 N29:5 BND OTE B13:13/0 EOR
%   B3:29/15  AFI %
%   N17:3  PT2211PI  "PRESSAO GIRO CANHAO" %
%   N16:27  PT2211HH  "GIRO CANHAO PRESSAO MUITO ALTA" %
%   B13:13/0  PT2211PTAHH  "PRESSAO GIRO CANHAO ALARME MUITO ALTA" %
%   N29:5  LIM_AL_HH  "LIMITE PARA PERMITIR O REARME DO ALARME HH (MUITO ALTO)" %

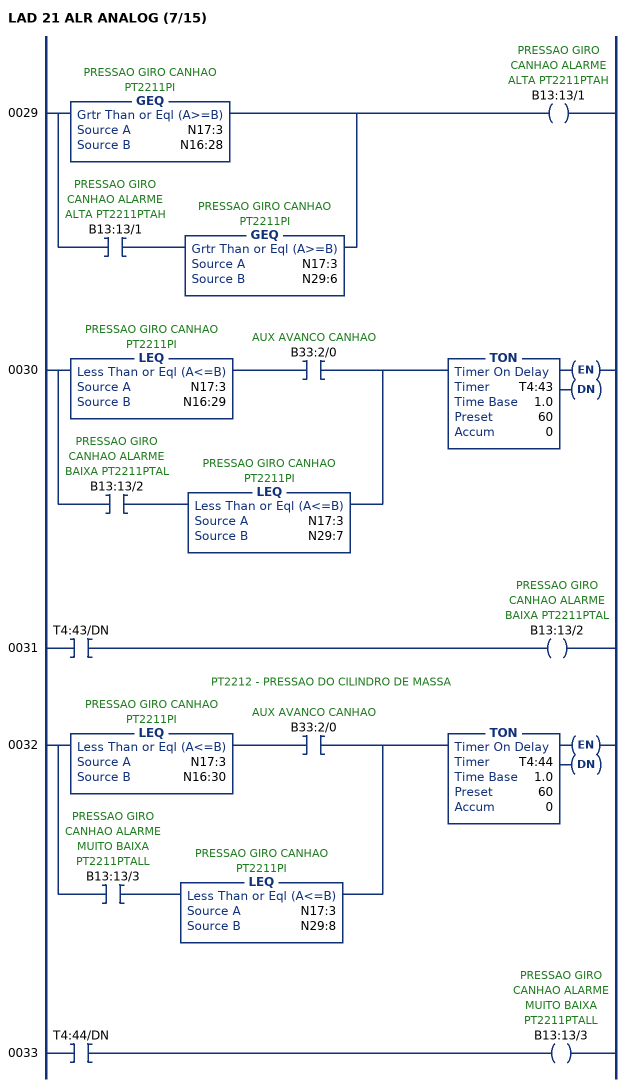
% Rung: 29 %
SOR BST GEQ N17:3 N16:28 NXB XIC B13:13/1 GEQ N17:3 N29:6 BND OTE B13:13/1 EOR
%   N17:3  PT2211PI  "PRESSAO GIRO CANHAO" %
%   N16:28  PT2211HF  "GIRO CANHAO PRESSAO ALTA" %
%   B13:13/1  PT2211PTAH  "PRESSAO GIRO CANHAO ALARME ALTA" %
%   N29:6  LIM_AL_H  "LIMITE PARA PERMITIR O REARME DO ALARME H (ALTO)" %
% Rung: 30 %
SOR BST LEQ N17:3 N16:29 XIC B33:2/0 NXB XIC B13:13/2 LEQ N17:3 N29:7 BND TON T4:43 1.0 60 0 EOR
%   N17:3  PT2211PI  "PRESSAO GIRO CANHAO" %
%   N16:29  PT2211L  "GIRO CANHAO PRESSAO BAIXA" %
%   B33:2/0  "AUX AVANCO CANHAO" %
%   B13:13/2  PT2211PTAL  "PRESSAO GIRO CANHAO ALARME BAIXA" %
%   N29:7  LIM_AL_L  "LIMITE PARA PERMITIR O REARME DO ALARME L (BAIXO)" %
% Rung: 31 %
SOR XIC T4:43/DN OTE B13:13/2 EOR
%   B13:13/2  PT2211PTAL  "PRESSAO GIRO CANHAO ALARME BAIXA" %
% Rung: 32 %
% PT2212 - PRESSAO DO CILINDRO DE MASSA %
SOR BST LEQ N17:3 N16:30 XIC B33:2/0 NXB XIC B13:13/3 LEQ N17:3 N29:8 BND TON T4:44 1.0 60 0 EOR
%   N17:3  PT2211PI  "PRESSAO GIRO CANHAO" %
%   N16:30  PT2211LL  "GIRO CANHAO PRESSAO MUITO BAIXA" %
%   B33:2/0  "AUX AVANCO CANHAO" %
%   B13:13/3  PT2211PTALL  "PRESSAO GIRO CANHAO ALARME MUITO BAIXA" %
%   N29:8  LIM_AL_LL  "LIMITE PARA PERMITIR O REARME DO ALARME LL (MUITO BAIXO)" %
% Rung: 33 %
SOR XIC T4:44/DN OTE B13:13/3 EOR
%   B13:13/3  PT2211PTALL  "PRESSAO GIRO CANHAO ALARME MUITO BAIXA" %

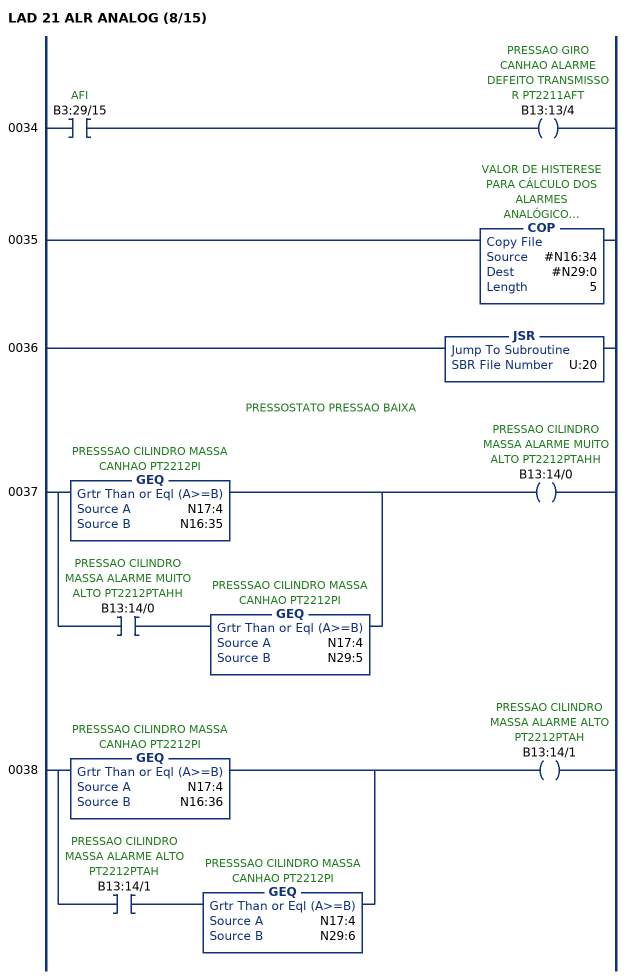
% Rung: 34 %
SOR XIC B3:29/15 OTE B13:13/4 EOR
%   B3:29/15  AFI %
%   B13:13/4  PT2211AFT  "PRESSAO GIRO CANHAO ALARME DEFEITO TRANSMISSOR" %
% Rung: 35 %
SOR COP #N16:34 #N29:0 5 EOR
%   N16:34  PT2212HIS  "CILINDRO MASSA CANHAO PRESSAO HISTERESE" %
%   N29:0  HISTERESE  "VALOR DE HISTERESE PARA CÁLCULO DOS ALARMES ANALÓGICOS" %
% Rung: 36 %
SOR JSR U:20 EOR
% Rung: 37 %
% PRESSOSTATO PRESSAO BAIXA %
SOR BST GEQ N17:4 N16:35 NXB XIC B13:14/0 GEQ N17:4 N29:5 BND OTE B13:14/0 EOR
%   N17:4  PT2212PI  "PRESSSAO CILINDRO MASSA CANHAO" %
%   N16:35  PT2212HH  "CILINDRO MASSA CANHAO PRESSAO MUITO ALTA" %
%   B13:14/0  PT2212PTAHH  "PRESSAO CILINDRO MASSA ALARME MUITO ALTO" %
%   N29:5  LIM_AL_HH  "LIMITE PARA PERMITIR O REARME DO ALARME HH (MUITO ALTO)" %
% Rung: 38 %
SOR BST GEQ N17:4 N16:36 NXB XIC B13:14/1 GEQ N17:4 N29:6 BND OTE B13:14/1 EOR
%   N17:4  PT2212PI  "PRESSSAO CILINDRO MASSA CANHAO" %
%   N16:36  PT2212H  "CILINDRO MASSA CANHAO PRESSAO ALTA" %
%   B13:14/1  PT2212PTAH  "PRESSAO CILINDRO MASSA ALARME ALTO" %
%   N29:6  LIM_AL_H  "LIMITE PARA PERMITIR O REARME DO ALARME H (ALTO)" %

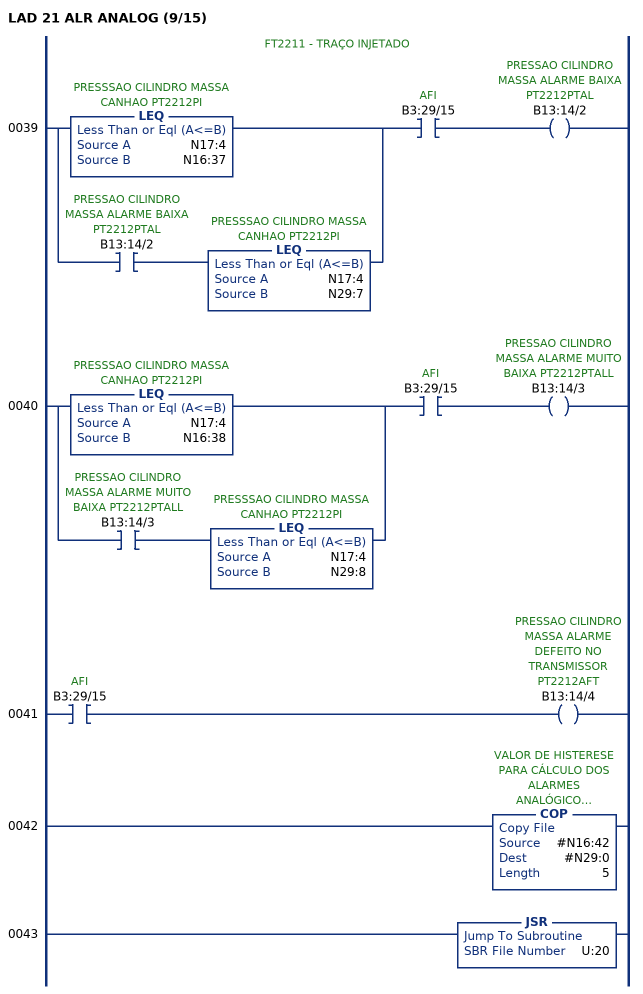
% Rung: 39 %
% FT2211 - TRAÇO INJETADO %
SOR BST LEQ N17:4 N16:37 NXB XIC B13:14/2 LEQ N17:4 N29:7 BND XIC B3:29/15 OTE B13:14/2 EOR
%   N17:4  PT2212PI  "PRESSSAO CILINDRO MASSA CANHAO" %
%   N16:37  PT2212L  "CILINDRO MASSA CANHAO PRESSAO BAIXA" %
%   B13:14/2  PT2212PTAL  "PRESSAO CILINDRO MASSA ALARME BAIXA" %
%   N29:7  LIM_AL_L  "LIMITE PARA PERMITIR O REARME DO ALARME L (BAIXO)" %
%   B3:29/15  AFI %
% Rung: 40 %
SOR BST LEQ N17:4 N16:38 NXB XIC B13:14/3 LEQ N17:4 N29:8 BND XIC B3:29/15 OTE B13:14/3 EOR
%   N17:4  PT2212PI  "PRESSSAO CILINDRO MASSA CANHAO" %
%   N16:38  PT2212LL  "CILINDRO MASSA CANHAO PRESSAO MUITO BAIXA" %
%   B13:14/3  PT2212PTALL  "PRESSAO CILINDRO MASSA ALARME MUITO BAIXA" %
%   N29:8  LIM_AL_LL  "LIMITE PARA PERMITIR O REARME DO ALARME LL (MUITO BAIXO)" %
%   B3:29/15  AFI %
% Rung: 41 %
SOR XIC B3:29/15 OTE B13:14/4 EOR
%   B3:29/15  AFI %
%   B13:14/4  PT2212AFT  "PRESSAO CILINDRO MASSA ALARME DEFEITO NO TRANSMISSOR" %
% Rung: 42 %
SOR COP #N16:42 #N29:0 5 EOR
%   N16:42  FT2211HIS  "TRACO INJETADO VAZAO HISTERESE" %
%   N29:0  HISTERESE  "VALOR DE HISTERESE PARA CÁLCULO DOS ALARMES ANALÓGICOS" %
% Rung: 43 %
SOR JSR U:20 EOR

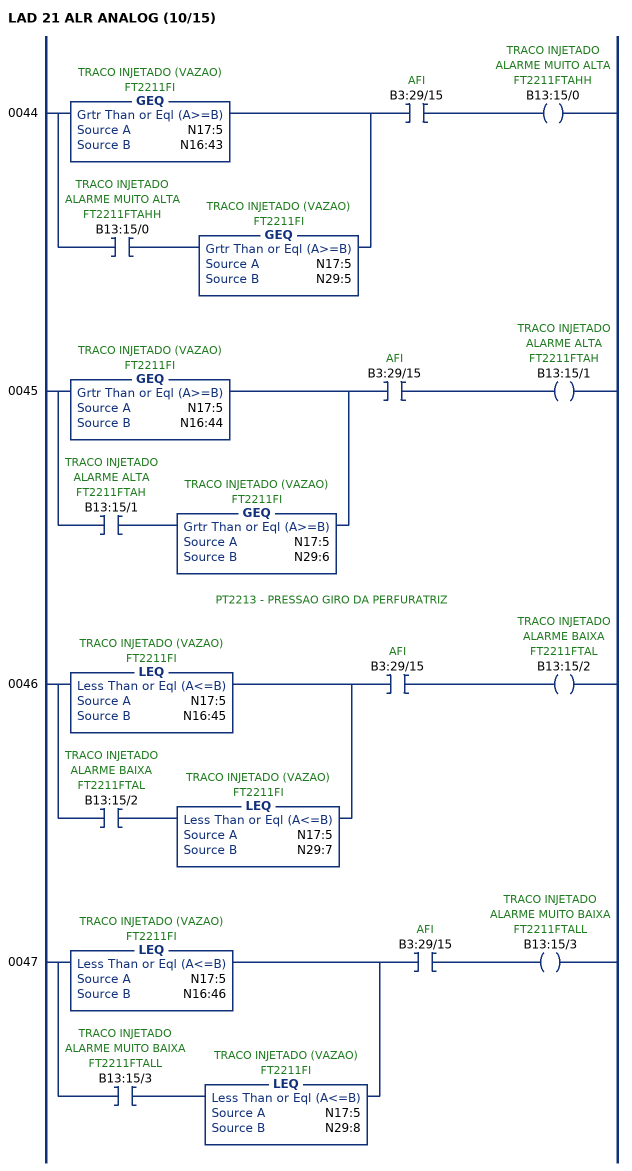
% Rung: 44 %
SOR BST GEQ N17:5 N16:43 NXB XIC B13:15/0 GEQ N17:5 N29:5 BND XIC B3:29/15 OTE B13:15/0 EOR
%   N17:5  FT2211FI  "TRACO INJETADO (VAZAO)" %
%   N16:43  FT2211HH  "TRACO INJETADO VAZAO MUITO ALTA" %
%   B13:15/0  FT2211FTAHH  "TRACO INJETADO ALARME MUITO ALTA" %
%   N29:5  LIM_AL_HH  "LIMITE PARA PERMITIR O REARME DO ALARME HH (MUITO ALTO)" %
%   B3:29/15  AFI %
% Rung: 45 %
SOR BST GEQ N17:5 N16:44 NXB XIC B13:15/1 GEQ N17:5 N29:6 BND XIC B3:29/15 OTE B13:15/1 EOR
%   N17:5  FT2211FI  "TRACO INJETADO (VAZAO)" %
%   N16:44  FT2211H  "TRACO INJETADO VAZAO ALTA" %
%   B13:15/1  FT2211FTAH  "TRACO INJETADO ALARME ALTA" %
%   N29:6  LIM_AL_H  "LIMITE PARA PERMITIR O REARME DO ALARME H (ALTO)" %
%   B3:29/15  AFI %
% Rung: 46 %
% PT2213 - PRESSAO GIRO DA PERFURATRIZ %
SOR BST LEQ N17:5 N16:45 NXB XIC B13:15/2 LEQ N17:5 N29:7 BND XIC B3:29/15 OTE B13:15/2 EOR
%   N17:5  FT2211FI  "TRACO INJETADO (VAZAO)" %
%   N16:45  FT2211L  "TRACO INJETADO VAZAO BAIXA" %
%   B13:15/2  FT2211FTAL  "TRACO INJETADO ALARME BAIXA" %
%   N29:7  LIM_AL_L  "LIMITE PARA PERMITIR O REARME DO ALARME L (BAIXO)" %
%   B3:29/15  AFI %
% Rung: 47 %
SOR BST LEQ N17:5 N16:46 NXB XIC B13:15/3 LEQ N17:5 N29:8 BND XIC B3:29/15 OTE B13:15/3 EOR
%   N17:5  FT2211FI  "TRACO INJETADO (VAZAO)" %
%   N16:46  FT2211LL  "TRACO INJETADO VAZAO MUITO BAIXA" %
%   B13:15/3  FT2211FTALL  "TRACO INJETADO ALARME MUITO BAIXA" %
%   N29:8  LIM_AL_LL  "LIMITE PARA PERMITIR O REARME DO ALARME LL (MUITO BAIXO)" %
%   B3:29/15  AFI %

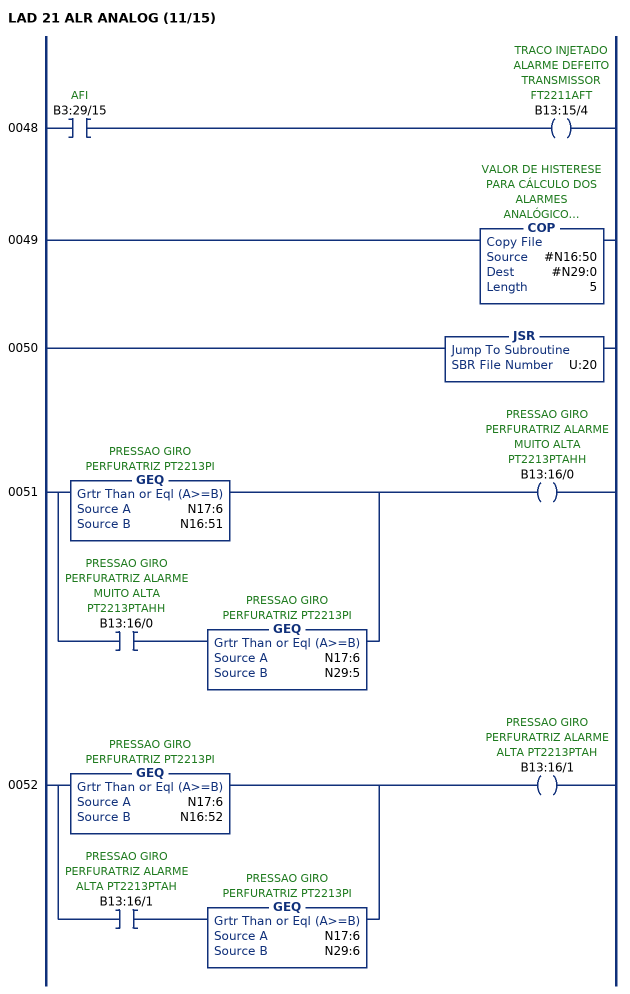
% Rung: 48 %
SOR XIC B3:29/15 OTE B13:15/4 EOR
%   B3:29/15  AFI %
%   B13:15/4  FT2211AFT  "TRACO INJETADO ALARME DEFEITO TRANSMISSOR" %
% Rung: 49 %
SOR COP #N16:50 #N29:0 5 EOR
%   N16:50  PT2213HIS  "PRESSAO GIRO PERFURATRIZ HISTERESE" %
%   N29:0  HISTERESE  "VALOR DE HISTERESE PARA CÁLCULO DOS ALARMES ANALÓGICOS" %
% Rung: 50 %
SOR JSR U:20 EOR
% Rung: 51 %
SOR BST GEQ N17:6 N16:51 NXB XIC B13:16/0 GEQ N17:6 N29:5 BND OTE B13:16/0 EOR
%   N17:6  PT2213PI  "PRESSAO GIRO PERFURATRIZ" %
%   N16:51  PT2213HH  "PRESSAO GIRO PERFURATRIZ MUITO ALTA" %
%   B13:16/0  PT2213PTAHH  "PRESSAO GIRO PERFURATRIZ ALARME MUITO ALTA" %
%   N29:5  LIM_AL_HH  "LIMITE PARA PERMITIR O REARME DO ALARME HH (MUITO ALTO)" %
% Rung: 52 %
SOR BST GEQ N17:6 N16:52 NXB XIC B13:16/1 GEQ N17:6 N29:6 BND OTE B13:16/1 EOR
%   N17:6  PT2213PI  "PRESSAO GIRO PERFURATRIZ" %
%   N16:52  PT2213H  "PRESSAO GIRO PERFURATRIZ ALTA" %
%   B13:16/1  PT2213PTAH  "PRESSAO GIRO PERFURATRIZ ALARME ALTA" %
%   N29:6  LIM_AL_H  "LIMITE PARA PERMITIR O REARME DO ALARME H (ALTO)" %

